# B&R Automation Studio project TD52 (part 125)

#### Ctr_HWSuCyclic.st
```iecst
(*******************************************************************************
Ctr_HWSu		controller heat water supply temperature

This code is confidential and proprietary to the INNIO Company.
It may not be used in any form, or reproduced in any manner,
without the express written permission of the INNIO Company.
Copyright, INNIO Company, 2022

Customized modifications: -
------------------------

History:
-------
V0.00.0		17.04.2012	lettenb.	Created
V3.99.0		23.11.2012	lettenb.	write back to IN_struct added (zengerer)
									tCtr_HWSu_In.Y_set := 100.0 -> 1.0, bugfix
V4.00.0		15.12.2014	lettenb.	controller interfaces completed like standard
V4.11.0		28.01.2022	Perktold	included plant controller upgrade

Instructions for use:
--------------------

Outstandings:
------------
(*******************************************************************************)

PROGRAM _CYCLIC

	(* Parameter *)
	Para.tCtr_HWSu.W_set;
	Para.tCtr_HWSu.W_set2;
	Para.tCtr_HWSu.W_min;
	Para.tCtr_HWSu.W_max;
	Para.tCtr_HWSu.dW_up;
	Para.tCtr_HWSu.dW_down;
	Para.tCtr_HWSu.deadband;
	Para.tCtr_HWSu.Y_min;
	Para.tCtr_HWSu.Y_max;
	Para.tCtr_HWSu.dY_max;
	Para.tCtr_HWSu.Y_block;
	Para.tCtr_HWSu.invert;
	Para.tCtr_HWSu.Kp;
	Para.tCtr_HWSu.Tn;
	Para.tCtr_HWSu.Tv;
	Para.tCtr_HWSu.Kp_GainScheduling;
	Para.tCtr_HWSu.Tn_GainScheduling;
	Para.tCtr_HWSu.Tv_GainScheduling;
	Para.tCtr_HWSu.t_min_pulse_down;
	Para.tCtr_HWSu.t_min_pulse_up;
	Para.tCtr_HWSu.t_period_down;
	Para.tCtr_HWSu.t_period_up;

	(* Input variables *)
	tCtr_HWSu_In				:= VIS2MM.tCtr_HWSu_In;			(* from vis *)

	(* Input from module *)
	tCtr_HWSu_In.enable			:=	Para.bCtr_HWSu
								AND	IN_HC.tPB2MM.bParaSetupOk
								AND IN_HC.bEng_Aux_Dem_CDR
								AND IN_HC.tT_HW_Su.GoodQual;
	tCtr_HWSu_In.W_ext_Active	:= tCtr_HWSu_In.W_ext_Active;	(* from vis *)
	tCtr_HWSu_In.W_ext			:= 0.0;
	tCtr_HWSu_In.Y_set_Active	:= NOT IN_HC.tT_HW_Su.GoodQual;
	tCtr_HWSu_In.Y_set			:= 1.0;
	tCtr_HWSu_In.X				:= IN_HC.tT_HW_Su.Ai;
	tCtr_HWSu_In.A				:= 0;
	tCtr_HWSu_In.W_set2_Active	:= FALSE;	(*Input to define which internal setpoint will be used TRUE = use the 2nd set point | FALSE use the normal "1st" one*)
	tCtr_HWSu_In.GainScheduling	:= 0.0;		(*Input for Gain Scheduling: 0.0 = use 100% of the Standard PID-Parameters | 1.0 = use 100% of the GainSched. PID Parameters | linear interpolation in between*)
	tCtr_HWSu_In.Y_min_cust		:= -1.0;	(*"customized" Y-Min at the current moment (The existing Y-Min parameter is the global minimum. To have an effect Y_min_cust needs to be > the parameter | -1.0 = function not used*)
	tCtr_HWSu_In.Y_max_cust		:= 1.0;		(*"customized" Y-Max at the current moment (The existing Y-Max parameter is the global maximum. To have an effect Y_max_cust needs to be < the parameter | 1.0 = function not used*)
	tCtr_HWSu_In.Retrigger		:= FALSE;	(*a rising edge on this input signals the controller to retrigger - set W on X and force the Integrator to the current Y*)

	(* Input from Visualization via OPC *)
	tCtr_HWSu_In.Y_man_Active;
	tCtr_HWSu_In.Y_man;
	tCtr_HWSu_In.X_min;
	tCtr_HWSu_In.X_max;
	tCtr_HWSu_In.Tune_quality;
	tCtr_HWSu_In.Tune_PI;
	tCtr_HWSu_In.Tune_PID;
	tCtr_HWSu_In.Tune_start;
	tCtr_HWSu_In.Tune_stop;
	tCtr_HWSu_In.Tune_takeover;

	xCtr_HWSu();

	(* Output variables function block *)
	(* Output to module(s) *)
	OUT_HC.tCtr_HWSu_Set.Ao 	:= tCtr_HWSu_Out.Y;	(* analog out *)

	(* Output to Visualization via OPC *)
	MM2VIS.tCtr_HWSu_Out		:= tCtr_HWSu_Out;
	VIS2MM.tCtr_HWSu_In			:= tCtr_HWSu_In;	(* write back to IN_struct for reset: Tune_takeover, X-display, ...!*)

	tCtr_HWSu_Out.Active;
	tCtr_HWSu_Out.Y;
	tCtr_HWSu_Out.W;
	tCtr_HWSu_Out.e;
	tCtr_HWSu_Out.Kp_tune;
	tCtr_HWSu_Out.Tn_tune;
	tCtr_HWSu_Out.Tv_tune;
	tCtr_HWSu_Out.status;

END_PROGRAM
```

#### Ctr_HWSuInit.st
```iecst
PROGRAM _INIT

	xCtr_HWSu.pParameter := ADR(Para.tCtr_HWSu);
	xCtr_HWSu.pInput 	 := ADR(tCtr_HWSu_In);
	xCtr_HWSu.pOutput	 := ADR(tCtr_HWSu_Out);

	tCtr_HWSu_In.AlwaysUseYRamp		:= TRUE;	(*If TRUE the Y signal will always limit the change rate via the according parameter | if FALSE the Y signal will jump in case the controller is disabled (blocked or set)*)
	tCtr_HWSu_In.KeepYManAtBlock	:= TRUE;	(*If TRUE the controller will keep the Y-man value constant in case the controller is disabled (blocked or set) | If FALSE the blocked or set value will override the Y-man value*)
	tCtr_HWSu_In.Y_min_cust			:= -1.0;	(*"customized" Y-Min at the current moment (The existing Y-Min parameter is the global minimum. To have an effect Y_min_cust needs to be > the parameter | -1.0 = function not used*)
	tCtr_HWSu_In.Y_max_cust			:=  1.0;	(*"customized" Y-Max at the current moment (The existing Y-Max parameter is the global maximum. To have an effect Y_max_cust needs to be < the parameter | 1.0 = function not used*)
	tCtr_HWSu_In.StepperMode		:= FALSE;	(* TRUE = use PWM-Mode (standard mode until 4.10) | FALSE = use continuous servo drive *)

END_PROGRAM
```

### Program Logical/HeatingCooling/MsgHC (IEC) - messages

#### MsgHCCyclic.st
```iecst
(*******************************************************************************
MsgHC	 			 messages

This code is confidential and proprietary to the INNIO Company.
It may not be used in any form, or reproduced in any manner,
without written permission of the INNIO Company.
Copyright, INNIO Company, 2025

Customized modifications: -
------------------------

History:
-------
V0.01.0	02.11.2011	lettenb.	new
V3.30.0 14.09.2011	lettenb.	2119 xTON_ChC_FanRdy added
V3.99.0	20.02.2013	lettenb.	3303,3521,3590 IN_HC.tT_HW_Re_LT.Ai added (V3.40)
		27.05.2013				3521 Para.bT_HW_Re_LT_Active added
		27.05.2013	Lettenb.	reset OUT_xx.txx2AB.bGnlTripx changed
		31.01.2014	lettenb.	1063 BWS_HA added(1063 NOT resetable in CASE OF sensor fail.)V350
V4.00.0	02.06.2014	lettenb.	3509 AND NOT MM2VIS.bMsg3312 added(hi-alarm in case of ms failure)
		16.06.2014	lettenb.	2104 xTP_2104, PT:= 0->1" added, acc.xt3 bugfix
V4.00.1 15.09.2014	lettenb.	1063 Para.bT_HW_Su_Active added
V4.00.2 17.11.2014				2638,2639,2640,2641,2647,2667 added, 920
								2104 enable with IN_HC.tPB2MM.bSys_Run
V4.00.3	19.03.2015				1021 STB active for 920+visa
		02.04.2015				2119 bugfix(portation failure from xt3)
V4.03.0 06.07.2015				920 ECW + EO module signals added(TCA redesign)
		25.07.2015	Plattner	2731-2736,2750,2751 failure boiler house ventilator added
		30.09.2015				2119 tAuxV_Aux_ok added
		17.03.2016	lettenb.	1021 KTMA_VISA added (920 umschaltung prio)
V4.04.0 07.04.2016	lettenb.	3492,3493,3494 added (TCA redesign2), 2640 disabled(double coded, 3590)
								2732,2734,2751 MS added + T#0s -> 2s, bugfix
		24.10.2016				2763 Functional Safety EN 13849
V4.05.0 27.02.2017	lettenb.	1032,1033 disabled for BR9 -> 2428,2429 added, SWAT920/1
		04.12.2017	Waldhart	1032,1033 enabled FOR BR9 -> 2428,2429 disabled, SWAT920/4
		22.12.2017	lettenb.	comment added: Safety-related application software source code (EN 13849-1 / 4.6.3)
		22.01.2018	lettenb.	1145,1186,1187,3407,3508,3526,3590 bParaSetupOk added TO avoid message at plc startup
V4.07.0	09.08.2018	Schmid		2nd low temperature charge cooling circuit added (W9226, W9228-W9232)
		08.10.2018	lettenb.	1063,1070,1071,1186,1187,2430,3312,3321,3508,3526,3590,9232 :bOMSS... removed, signal failure active in stop-mode
		11.10.2018	lettenb.	2720: enable Para.bT_Re_SecCirc_Active, bugfix
		17.12.2018	Schmid		OUT_HC.bMsg2684 -> AG vvm added
		06.06.2019	lettenb.	2733,2736,2752,3492,3493,3494 bParaSetupOk added to avoid alarm at plc-startup
V4.10.0	20.07.2020	Schmid		2341, 2342, 2343 additional heating water circuit monitoring
V4.11.0	17.01.2022	lettenb.	2736 delay 2s added, bugfix
V4.14.0 08.11.2024	Bacci		9098, 9099 added
		11.12.2024	Nagy		1019,1021,1050,3402 modified (2024-225)
V4.25.0	10.07.2025	Tinello		SafetyPLC: Added monitoring for heating water supply temperature unit W9588, W9589

Instructions for use:
--------------------
1) declare alarm with function block "Msg"
	declare buffert alarm bit bMsg<message number>

2) use template to create a new alarm,
   substitue 0000 by alarm number and make settings:

	xMsg0000.Enable		:=	TRUE;		enable/disable alarm
	xMsg0000.Set		:=	FALSE;		alarm set condition
	xMsg0000.PT			:=	T#0s;		alarm delay time
	xMsg0000.Prio		:=	1;			alarm priority: 1-3 = trip, 4 = warning
	xMsg0000.RiskClass	:=	3;			risk class for remote alarm reset acc.TI 1100-0111
	xMsg0000.Reset		:=	FALSE;		FALSE: for all standard alarms	prio 1,2,3 and warnings prio 4
										TRUE : for autoreset alarms

	bMsg0000			:=	xMsg0000.Q;	connect buffert alarm bit for VIS and control
	bMsg0000_Test		:=	xMsg0000.Test; alarm bypass active

3)  expand INIT

Outstandings:
------------
(*******************************************************************************)
PROGRAM _CYCLIC

	(* reset general trip *)
	OUT_HC.tHC2AB.bGnlTrip1		:=	FALSE;
	OUT_HC.tHC2AB.bGnlTrip2		:=	FALSE;
	OUT_HC.tHC2AB.bGnlTrip3		:=	FALSE;
	OUT_HC.tHC2AB.bGnlWarning	:=	FALSE;
	OUT_HC.tHC2AB.bTriptype1	:=	FALSE;
	OUT_HC.tHC2AB.bTriptype2	:=	FALSE;
	OUT_HC.tHC2AB.bTriptype3	:=	FALSE;

	(*---------------------------------------------------------------------------*)
	xTON_EngRunAnd10s(IN:= IN_HC.tEng_Run.Do, PT:= T#10s);
	xTON_EngRunAnd60s(IN:= IN_HC.tEng_Run.Do, PT:= T#60s);

	(********************************************************************************************************************
	Safety-related application software source code (EN 13849-1 / 4.6.3): BEGIN
	*********************************************************************************************************************)

	(*  1019 engine cooling water pressure low *)
	xTP_1019(IN:= IN_HC.tECWP1Dem.Do, PT:= T#10s);	(* lock monitoring *)

	xMsg1019.Enable		:=	TRUE;
	xMsg1019.Set		:=	(bPr_ECW_LoLo OR bPr_ECW_LoLoPrio2) AND NOT xTP_1019.Q;
	xMsg1019.PT			:=	T#0s;
	IF bPr_ECW_LoLoPrio2 THEN
		xMsg1019.Prio		:=	2;
	ELSE
		xMsg1019.Prio		:=	3;
	END_IF;
	xMsg1019.RiskClass	:=	10;
	xMsg1019.Reset		:=	FALSE;
	xMsg1019();
	MM2VIS.bMsg1019     := xMsg1019.Q;
	OUT_HC.bMsg1019     := xMsg1019.Q;

	(********************************************************************************************************************
	Safety-related application software source code (EN 13849-1 / 4.6.3): END
	*********************************************************************************************************************)

	(* A1021 engine cooling water temperature high *)
	xTON_1021(IN:= OUT_HC.bT_ECW_Hi, PT:= T#2h);

	xMsg1021.Enable		:=	TRUE;
	xMsg1021.Set		:= ((xTON_1021.Q OR bT_ECW_HiHi OR bT_ECW_HiHiPrio2) AND xTON_EngRunAnd60s.Q AND NOT MM2VIS.bMsg2101)
						OR  IN_HC.tT_ECW_Ext_Hi.Di; (*STB: VISA + 920*)
	xMsg1021.PT			:=	T#0s;
	KTMA_VISA := IN_HC.tT_ECW_Ext_Hi.Di OR (KTMA_VISA AND xMsg1021.Q);
	IF (Para.bVISA OR xEngType.Type9) AND KTMA_VISA OR bT_ECW_HiHiPrio2 THEN	(* umschaltung prio nur bei abstellung durch STB(sicherheitsschleife) *)
		xMsg1021.Prio	:=	2;
	ELSE
		xMsg1021.Prio	:=	3;
	END_IF;
	xMsg1021.RiskClass	:=	0;
	xMsg1021.Reset		:=	FALSE;
	xMsg1021();
	MM2VIS.bMsg1021     := xMsg1021.Q;

	(* A1032 heat water flow low (W2428)*)
	xTOF_EngDemEPS(IN:= IN_HC.bEng_Dem_EPS AND NOT IN_HC.tGCB_On.Di, PT:= T#60s);
	bNoMon4BlackStart := xTOF_EngDemEPS.Q AND IN_HC.bEng_Dem_EPS; //T14

	xMsg1032.Enable		:=	TRUE;//SWAT920/4
	xMsg1032.Set 		:=	NOT IN_HC.tFlow_HW_Lo.Di
						AND NOT bNoMon4BlackStart AND IN_HC.tEng_Run.Do;
	xMsg1032.PT			:=	T#10s;
	xMsg1032.Prio		:=	3;
	xMsg1032.RiskClass	:=	4;
	xMsg1032.Reset		:=	FALSE;
	xMsg1032();
	MM2VIS.bMsg1032     := xMsg1032.Q;

	(* A1033 heat water temperature high (W2429)*)
	xMsg1033.Enable		:=	TRUE;//SWAT920/4
	xMsg1033.Set 		:=	IN_HC.tT_HW_Hi.Di OR IN_HC.tT_HW_Hi1.Di;
	xMsg1033.PT			:=	T#0s;
	xMsg1033.Prio		:=	2;
	xMsg1033.RiskClass	:=	4;
	xMsg1033.Reset		:=	FALSE;
	xMsg1033();
	MM2VIS.bMsg1033     := xMsg1033.Q;

	(* A1034 heat water pressure low *)
	xMsg1034.Enable		:=	TRUE;
	xMsg1034.Set 		:=  IN_HC.tPr_HW_Lo.Di;
	xMsg1034.PT			:=	T#0s;
	xMsg1034.Prio		:=	2;
	xMsg1034.RiskClass	:=	4;
	xMsg1034.Reset		:=	FALSE;
	xMsg1034();
	MM2VIS.bMsg1034     := xMsg1034.Q;

	(* A1035 heat water pressure high *)
	xMsg1035.Enable		:=	TRUE;
	xMsg1035.Set 		:=  IN_HC.tPr_HW_Hi.Di OR IN_HC.tPr_HW_Hi1.Di;
	xMsg1035.PT			:=	T#0s;
	xMsg1035.Prio		:=	2;
	xMsg1035.RiskClass	:=	4;
	xMsg1035.Reset		:=	FALSE;
	xMsg1035();
	MM2VIS.bMsg1035     := xMsg1035.Q;

	(* A1050 engine cooling water pressure high *)
	(* lock monitoring jacket water pressure high at engine start. (reference: W3406)
	(in case of rising jacket water pressure with rising oil pressure.
	caused by pressure transfered from oil circuit to water circuit by the plate heat exchanger)*)
	xTP_1050(IN:= bN_EngStart, PT:= T#20s);

	xMsg1050.Enable		:=	TRUE;
	xMsg1050.Set := (bPr_ECW_HiHi OR bPr_ECW_HiHiPrio2) AND NOT xTP_1050.Q;
	xMsg1050.PT			:=	T#0s;
	IF bPr_ECW_HiHiPrio2 THEN
		xMsg1050.Prio		:=	2;
	ELSE
		xMsg1050.Prio		:=	3;
	END_IF;
	xMsg1050.RiskClass	:=	2;
	xMsg1050.Reset		:=	FALSE;
	xMsg1050();
	MM2VIS.bMsg1050     := xMsg1050.Q;
	OUT_HC.bMsg1050		:= xMsg1050.Q;

	(* A1063 heat water supply temperature high (W2430)*)
	xMsg1063.Enable		:=	Para.bT_HW_Su_Active;
	xMsg1063.Set 		:=  bT_HW_Su_HiHi AND NOT MM2VIS.bMsg1071 AND NOT MM2VIS.bMsg1187;
	xMsg1063.PT			:=	T#2s;
	xMsg1063.Prio		:=	3;
	xMsg1063.RiskClass	:=	0;
	xMsg1063.Reset		:=	FALSE;
	xMsg1063();
	MM2VIS.bMsg1063     := xMsg1063.Q;

	(* A1070 heat water return temperature signal failure trip (W1186)*)
	xMsg1070.Enable		:=	Para.bT_HW_Re_Active AND Para.bT_HW_Re_SF_Trip;
	xMsg1070.Set 		:=	NOT IN_HC.tT_HW_Re.GoodQual;
	xMsg1070.PT			:=	T#0s;
	xMsg1070.Prio		:=	3;
	xMsg1070.RiskClass	:=	4;
	xMsg1070.Reset		:=	FALSE;
	xMsg1070();
	MM2VIS.bMsg1070     := xMsg1070.Q;

	(* A1071 heat water supply temperature signal failure trip (W1187)*)
	xMsg1071.Enable		:=	Para.bT_HW_Su_Active AND Para.bT_HW_Su_SF_Trip;
	xMsg1071.Set 		:=  NOT IN_HC.tT_HW_Su.GoodQual;
	xMsg1071.PT			:=	T#0s;
	xMsg1071.Prio		:=	3;
	xMsg1071.RiskClass	:=	4;
	xMsg1071.Reset		:=	FALSE;
	xMsg1071();
	MM2VIS.bMsg1071     := xMsg1071.Q;

	(* A1130 charge cooler water pressure low (W2117)*)
	xMsg1130.Enable		:=	FALSE;
	xMsg1130.Set		:=	NOT IN_HC.tPr_ChC_Lo.Di;
	xMsg1130.PT			:=	T#0s;
	xMsg1130.Prio		:=	3;
	xMsg1130.RiskClass	:=	4;
	xMsg1130.Reset		:=	FALSE;
	xMsg1130();
	MM2VIS.bMsg1130     := xMsg1130.Q;

	(* W1145 engine cooling water temperature low *)
	xMsg1145.Enable		:=	IN_HC.tPB2MM.bParaSetupOk;
	xMsg1145.Set 		:=  OUT_HC.bT_ECW_Lo;
	xMsg1145.PT			:=	T#0s;
	xMsg1145.Prio		:=	4;
	xMsg1145.RiskClass	:=	4;
	xMsg1145.Reset		:=	FALSE;
	xMsg1145();
	MM2VIS.bMsg1145     := xMsg1145.Q;

	(* W1167  heat water return temperature high *)
	xTON_1167(IN:= NOT MM2VIS.bMsg1186 AND NOT MM2VIS.bMsg1070 AND bT_HW_Re_Hi, PT:= T#10s);

	xMsg1167.Enable		:=	Para.bT_HW_Re_Active;
	xMsg1167.Set 		:=  xTON_EngRunAnd10s.Q AND xTON_1167.Q;
	xMsg1167.PT			:=	T#0s;
	xMsg1167.Prio		:=	4;
	xMsg1167.RiskClass	:=	4;
	xMsg1167.Reset		:=	FALSE;
	xMsg1167();
	MM2VIS.bMsg1167     := xMsg1167.Q;

	(* W1186 heat water return temperature signal failure (A1070)*)
	xMsg1186.Enable		:=	Para.bT_HW_Re_Active AND NOT Para.bT_HW_Re_SF_Trip AND IN_HC.tPB2MM.bParaSetupOk;
	xMsg1186.Set 		:=  NOT IN_HC.tT_HW_Re.GoodQual;
	xMsg1186.PT			:=	T#0s;
	xMsg1186.Prio		:=	4;
	xMsg1186.RiskClass	:=	4;
	xMsg1186.Reset		:=	FALSE;
	xMsg1186();
	MM2VIS.bMsg1186     := xMsg1186.Q;

	(* W1187 heat water supply temperature signal failure (A1071)*)
	xMsg1187.Enable		:=	Para.bT_HW_Su_Active AND NOT Para.bT_HW_Su_SF_Trip AND IN_HC.tPB2MM.bParaSetupOk;
	xMsg1187.Set 		:=  NOT IN_HC.tT_HW_Su.GoodQual;
	xMsg1187.PT			:=	T#0s;
	xMsg1187.Prio		:=	4;
	xMsg1187.RiskClass	:=	4;
	xMsg1187.Reset		:=	FALSE;
	xMsg1187();
	MM2VIS.bMsg1187     := xMsg1187.Q;

	(* W2101 engine cooling water temperature signal failure *)
	xMsg2101.Enable		:=	TRUE;
	xMsg2101.Set		:= (NOT IN_HC.tT_ECW.GoodQual AND IN_HC.tPB2MM.bParaSetupOk)
						OR (xMsg2101.Set AND IN_HC.bMsg3003 AND bOMSS_MAT);
	xMsg2101.PT			:=	T#0s;
	xMsg2101.Prio		:=	4;
	xMsg2101.RiskClass	:=	4;
	xMsg2101.Reset		:=	FALSE;
	xMsg2101();
	MM2VIS.bMsg2101     := xMsg2101.Q;
	OUT_HC.bMsg2101     := xMsg2101.Q;

	(********************************************************************************************************************
	Safety-related application software source code (EN 13849-1 / 4.6.3): BEGIN
	*********************************************************************************************************************)
	(* W2104 engine cooling water pressure signal failure *)
	xTP_2104(IN:= IN_HC.tECWP1Dem.Do, PT:= T#10s);	(* lock monitoring *)

	xMsg2104.Enable		:=	IN_HC.tPB2MM.bSys_Run;
	xMsg2104.Set		:= (NOT IN_HC.tPr_ECW.GoodQual AND NOT xTP_2104.Q)
						OR (xMsg2104.Set AND IN_HC.bMsg3003 AND bOMSS_MAT);
	xMsg2104.PT			:=	T#1s;
	xMsg2104.Prio		:=	4;
	xMsg2104.RiskClass	:=	4;
	xMsg2104.Reset		:=	FALSE;
	xMsg2104();
	MM2VIS.bMsg2104     := xMsg2104.Q;
	OUT_HC.bMsg2104     := xMsg2104.Q;
	(********************************************************************************************************************
	Safety-related application software source code (EN 13849-1 / 4.6.3): END
	*********************************************************************************************************************)

	(* W2116 emergency cooler failure *)
	xMsg2116.Enable		:=	TRUE;
	xMsg2116.Set		:=	NOT IN_HC.tEC_Failure.Di AND NOT bNoMon4BlackStart;
	xMsg2116.PT			:=	T#0s;
	xMsg2116.Prio		:=	4;
	xMsg2116.RiskClass	:=	4;
	xMsg2116.Reset		:=	FALSE;
	xMsg2116();
	MM2VIS.bMsg2116     := xMsg2116.Q;

	(* W2117 charge cooler water pressure low (A1130)*)
	xMsg2117.Enable		:=	TRUE;
	xMsg2117.Set		:=	NOT IN_HC.tPr_ChC_Lo.Di;
	xMsg2117.PT			:=	T#10s;
	xMsg2117.Prio		:=	4;
	xMsg2117.RiskClass	:=	4;
	xMsg2117.Reset		:=	FALSE;
	xMsg2117();
	MM2VIS.bMsg2117     := xMsg2117.Q;
	OUT_HC.bMsg2117     := xMsg2117.Q;

	(* W2119 charge cooler failure *)
	xTON_ChC_FanRdy(IN:= (IN_HC.tAuxV_Supply_Ok.Di AND IN_HC.tAuxV_Aux_ok.Di) AND NOT IN_HC.tChC_FanRdy.Di, PT:= T#10s);		(*PJ*)

	xMsg2119.Enable		:=	TRUE;
	xMsg2119.Set		:=	NOT bNoMon4BlackStart AND(xTON_ChC_FanRdy.Q OR NOT IN_HC.tChC_Failure.Di);
	xMsg2119.PT			:=	T#0s;
	xMsg2119.Prio		:=	4;
	xMsg2119.RiskClass	:=	4;
	xMsg2119.Reset		:=	FALSE;
	xMsg2119();
	MM2VIS.bMsg2119     := xMsg2119.Q;

	(* A2341 Heating water temperature maximum - exhaust gas cooler *)
	xMsg2341.Enable		:=	IN_HC.tT_HW_EGHE_Hi.GoodQual;
	xMsg2341.Set 		:=	IN_HC.tT_HW_EGHE_Hi.Di;
	xMsg2341.PT			:=	T#0s;
	xMsg2341.Prio		:=	2;
	xMsg2341.RiskClass	:=	4;
	xMsg2341.Reset		:=	FALSE;
	xMsg2341();
	MM2VIS.bMsg2341     := xMsg2341.Q;

	(* A2342 Heating water temperature maximum - exhaust gas condenser *)
	xMsg2342.Enable		:=	IN_HC.tT_HW_EGCD_Hi.GoodQual;
	xMsg2342.Set 		:=	IN_HC.tT_HW_EGCD_Hi.Di;
	xMsg2342.PT			:=	T#0s;
	xMsg2342.Prio		:=	2;
	xMsg2342.RiskClass	:=	4;
	xMsg2342.Reset		:=	FALSE;
	xMsg2342();
	MM2VIS.bMsg2342     := xMsg2342.Q;

	(* A2343 External heating water circuit monitoring tripped *)
	xMsg2343.Enable		:=	IN_HC.tCust_HW_Ext_Trip.GoodQual;
	xMsg2343.Set 		:=	IN_HC.tCust_HW_Ext_Trip.Di;
	xMsg2343.PT			:=	T#0s;
	xMsg2343.Prio		:=	2;
	xMsg2343.RiskClass	:=	4;
	xMsg2343.Reset		:=	FALSE;
	xMsg2343();
	MM2VIS.bMsg2343     := xMsg2343.Q;

	(* W2428 heat water flow low (A1032)*)
	xMsg2428.Enable		:=	FALSE;//SWAT920/4
	xMsg2428.Set 		:=	NOT IN_HC.tFlow_HW_Lo.Di
						AND NOT bNoMon4BlackStart AND IN_HC.tEng_Run.Do;
	xMsg2428.PT			:=	T#10s;
	xMsg2428.Prio		:=	4;
	xMsg2428.RiskClass	:=	4;
	xMsg2428.Reset		:=	FALSE;
	xMsg2428();
	MM2VIS.bMsg2428     := xMsg2428.Q;

	(* W2429 heat water temperature high (A1033)*)
	xMsg2429.Enable		:=	FALSE;//SWAT920/4
	xMsg2429.Set 		:=	IN_HC.tT_HW_Hi.Di OR IN_HC.tT_HW_Hi1.Di;
	xMsg2429.PT			:=	T#0s;
	xMsg2429.Prio		:=	4;
	xMsg2429.RiskClass	:=	4;
	xMsg2429.Reset		:=	FALSE;
	xMsg2429();
	MM2VIS.bMsg2429     := xMsg2429.Q;

	(* W2430 heat water supply temperature high (A1063)*)//SWAT920/1
	xMsg2430.Enable		:=	Para.bT_HW_Su_Active;
	xMsg2430.Set 		:=  bT_HW_Su_Hi AND NOT MM2VIS.bMsg1071 AND NOT MM2VIS.bMsg1187;
	xMsg2430.PT			:=	T#2s;
	xMsg2430.Prio		:=	4;
	xMsg2430.RiskClass	:=	0;
	xMsg2430.Reset		:=	FALSE;
	xMsg2430();
	MM2VIS.bMsg2430     := xMsg2430.Q;

	(* W2638 heat water supply pressure LT circuit signal failure *)
	xMsg2638.Enable		:=	Para.bPr_HW_Su_LT_Active;
	xMsg2638.Set		:=	IN_HC.tPB2MM.bParaSetupOk AND NOT IN_HC.tPr_HW_Su_LT.GoodQual;
	xMsg2638.PT			:=	T#0s;
	xMsg2638.Prio		:=	4;
	xMsg2638.RiskClass	:=	4;
	xMsg2638.Reset		:=	FALSE;
	xMsg2638();
	MM2VIS.bMsg2638     := xMsg2638.Q;

	(* W2639 heat water supply pressure HT circuit signal failure *)
	xMsg2639.Enable		:=	Para.bPr_HW_Su_HT_Active;
	xMsg2639.Set		:=	IN_HC.tPB2MM.bParaSetupOk AND NOT IN_HC.tPr_HW_Su_HT.GoodQual;
	xMsg2639.PT			:=	T#0s;
	xMsg2639.Prio		:=	4;
	xMsg2639.RiskClass	:=	4;
	xMsg2639.Reset		:=	FALSE;
	xMsg2639();
	MM2VIS.bMsg2639     := xMsg2639.Q;

	(* W2640 heat water return temperature LT circuit signal failure *)(* -> 3590 *)
	xMsg2640.Enable		:=	Para.bT_HW_Re_LT_Active AND FALSE;
	xMsg2640.Set		:=	IN_HC.tPB2MM.bParaSetupOk AND NOT IN_HC.tT_HW_Re_LT.GoodQual;
	xMsg2640.PT			:=	T#0s;
	xMsg2640.Prio		:=	4;
	xMsg2640.RiskClass	:=	4;
	xMsg2640.Reset		:=	FALSE;
	xMsg2640();
	MM2VIS.bMsg2640     := xMsg2640.Q;

	(* W2641 heat water supply temperature LT circuit signal failure *)
	xMsg2641.Enable		:=	Para.bT_HW_Su_LT_Active;
	xMsg2641.Set		:=	IN_HC.tPB2MM.bParaSetupOk AND NOT IN_HC.tT_HW_Su_LT.GoodQual;
	xMsg2641.PT			:=	T#0s;
	xMsg2641.Prio		:=	4;
	xMsg2641.RiskClass	:=	4;
	xMsg2641.Reset		:=	FALSE;
	xMsg2641();
	MM2VIS.bMsg2641     := xMsg2641.Q;

	(* W2647 engine cooling water pressure after engine signal failure *)
	xMsg2647.Enable	   := Para.bPr_ECWaEng_Active;
	xMsg2647.Set       := IN_HC.tPB2MM.bParaSetupOk AND NOT IN_HC.tPr_ECWaEng.GoodQual;
	xMsg2647.PT		   := T#0s;
	xMsg2647.Prio	   := 4;
	xMsg2647.RiskClass := 4;
	xMsg2647.Reset	   := FALSE;
	xMsg2647();
	MM2VIS.bMsg2647	   := xMsg2647.Q;

	(* W2667 engine cooling water temperature before engine signal failure *)
	xMsg2667.Enable	   := Para.bT_ECWbEng_Active;
	xMsg2667.Set       := IN_HC.tPB2MM.bParaSetupOk AND NOT IN_HC.tT_ECWbEng.GoodQual;
	xMsg2667.PT		   := T#0s;
	xMsg2667.Prio	   := 4;
	xMsg2667.RiskClass := 4;
	xMsg2667.Reset	   := FALSE;
	xMsg2667();
	MM2VIS.bMsg2667	   := xMsg2667.Q;

	(* W2675 Pressure heat water return low temperature circuit return signal failure *)
	xMsg2675.Enable	   := Para.bPr_HW_Re_LT_Active;
	xMsg2675.Set       := IN_HC.tPB2MM.bParaSetupOk AND NOT IN_HC.tPr_HW_Re_LT.GoodQual;
	xMsg2675.PT		   := T#0s;
	xMsg2675.Prio	   := 4;
	xMsg2675.RiskClass := 4;
	xMsg2675.Reset	   := FALSE;
	xMsg2675();
	MM2VIS.bMsg2675	   := xMsg2675.Q;

	(* W2676 Pressure heat water return high temperature circuit signal failure *)
	xMsg2676.Enable	   := Para.bPr_HW_Re_HT_Active;
	xMsg2676.Set       := IN_HC.tPB2MM.bParaSetupOk AND NOT IN_HC.tPr_HW_Re_HT.GoodQual;
	xMsg2676.PT		   := T#0s;
	xMsg2676.Prio	   := 4;
	xMsg2676.RiskClass := 4;
	xMsg2676.Reset	   := FALSE;
	xMsg2676();
	MM2VIS.bMsg2676	   := xMsg2676.Q;

	(* W2677 Pressure heat water return hydraulic engine cooling water preheating signal failure *)
	xMsg2677.Enable	   := Para.bPr_HW_Re_PreH_ECW_Active;
	xMsg2677.Set       := IN_HC.tPB2MM.bParaSetupOk AND NOT IN_HC.tPr_HW_Re_PreH_ECW.GoodQual;
	xMsg2677.PT		   := T#0s;
	xMsg2677.Prio	   := 4;
	xMsg2677.RiskClass := 4;
	xMsg2677.Reset	   := FALSE;
	xMsg2677();
	MM2VIS.bMsg2677	   := xMsg2677.Q;

	(* W2678 Pressure heat water return hydraulic oil preheating signal failure *)
	xMsg2678.Enable	   := Para.bPr_HW_Re_PreH_EO_Active;
	xMsg2678.Set       := IN_HC.tPB2MM.bParaSetupOk AND NOT IN_HC.tPr_HW_Re_PreH_EO.GoodQual;
	xMsg2678.PT		   := T#0s;
	xMsg2678.Prio	   := 4;
	xMsg2678.RiskClass := 4;
	xMsg2678.Reset	   := FALSE;
	xMsg2678();
	MM2VIS.bMsg2678	   := xMsg2678.Q;

	(* W2679 Pressure oil module oil outlet signal failure *)
	xMsg2679.Enable	   := Para.bPr_EO_Mod_Out_Active;
	xMsg2679.Set       := IN_HC.tPB2MM.bParaSetupOk AND NOT IN_HC.tPr_EO_Mod_Out.GoodQual;
	xMsg2679.PT		   := T#0s;
	xMsg2679.Prio	   := 4;
	xMsg2679.RiskClass := 4;
	xMsg2679.Reset	   := FALSE;
	xMsg2679();
	MM2VIS.bMsg2679	   := xMsg2679.Q;

	(* W2680 Temperature engine cooling water module inlet  signal failure *)
	xMsg2680.Enable	   := Para.bT_ECW_Mod_In_Active;
	xMsg2680.Set       := IN_HC.tPB2MM.bParaSetupOk AND NOT IN_HC.tT_ECW_Mod_In.GoodQual;
	xMsg2680.PT		   := T#0s;
	xMsg2680.Prio	   := 4;
	xMsg2680.RiskClass := 4;
	xMsg2680.Reset	   := FALSE;
	xMsg2680();
	MM2VIS.bMsg2680	   := xMsg2680.Q;

	(* W2681 Temperature engine cooling water module outlet  signal failure *)
	xMsg2681.Enable	   := Para.bT_ECW_Mod_Out_Active;
	xMsg2681.Set       := IN_HC.tPB2MM.bParaSetupOk AND NOT IN_HC.tT_ECW_Mod_Out.GoodQual;
	xMsg2681.PT		   := T#0s;
	xMsg2681.Prio	   := 4;
	xMsg2681.RiskClass := 4;
	xMsg2681.Reset	   := FALSE;
	xMsg2681();
	MM2VIS.bMsg2681	   := xMsg2681.Q;

	(* W2682 Temperature oil module oil inlet signal failure *)
	xMsg2682.Enable	   := Para.bT_EO_Mod_In_Active;
	xMsg2682.Set       := IN_HC.tPB2MM.bParaSetupOk AND NOT IN_HC.tT_EO_Mod_In.GoodQual;
	xMsg2682.PT		   := T#0s;
	xMsg2682.Prio	   := 4;
	xMsg2682.RiskClass := 4;
	xMsg2682.Reset	   := FALSE;
	xMsg2682();
	MM2VIS.bMsg2682	   := xMsg2682.Q;

	(* W2683 Temperature oil module oil outlet  signal failure *)
	xMsg2683.Enable	   := Para.bT_EO_Mod_Out_Active;
	xMsg2683.Set       := IN_HC.tPB2MM.bParaSetupOk AND NOT IN_HC.tT_EO_Mod_Out.GoodQual;
	xMsg2683.PT		   := T#0s;
	xMsg2683.Prio	   := 4;
	xMsg2683.RiskClass := 4;
	xMsg2683.Reset	   := FALSE;
	xMsg2683();
	MM2VIS.bMsg2683	   := xMsg2683.Q;

	(* W2684 Temperature heat water supply hydraulic engine cooling water preheating signal failure *)
	xMsg2684.Enable	   := Para.bT_HW_Su_PreH_ECW_Active;
	xMsg2684.Set       := IN_HC.tPB2MM.bParaSetupOk AND NOT IN_HC.tT_HW_Su_PreH_ECW.GoodQual;
	xMsg2684.PT		   := T#0s;
	xMsg2684.Prio	   := 4;
	xMsg2684.RiskClass := 4;
	xMsg2684.Reset	   := FALSE;
	xMsg2684();
	MM2VIS.bMsg2684	   := xMsg2684.Q;
	OUT_HC.bMsg2684    := xMsg2684.Q;

	(* W2685 Temperature heat water return hydraulic engine cooling water preheating signal failure *)
	xMsg2685.Enable	   := Para.bT_HW_Re_PreH_ECW_Active;
	xMsg2685.Set       := IN_HC.tPB2MM.bParaSetupOk AND NOT IN_HC.tT_HW_Re_PreH_ECW.GoodQual;
	xMsg2685.PT		   := T#0s;
	xMsg2685.Prio	   := 4;
	xMsg2685.RiskClass := 4;
	xMsg2685.Reset	   := FALSE;
	xMsg2685();
	MM2VIS.bMsg2685	   := xMsg2685.Q;

	(* W2686 Temperature heat water supply hydraulic oil preheating signal failure *)
	xMsg2686.Enable	   := Para.bT_HW_Su_PreH_EO_Active;
	xMsg2686.Set       := IN_HC.tPB2MM.bParaSetupOk AND NOT IN_HC.tT_HW_Su_PreH_EO.GoodQual;
	xMsg2686.PT		   := T#0s;
	xMsg2686.Prio	   := 4;
	xMsg2686.RiskClass := 4;
	xMsg2686.Reset	   := FALSE;
	xMsg2686();
	MM2VIS.bMsg2686	   := xMsg2686.Q;

	(* W2687 Temperature heat water return hydraulic oil preheating signal failure *)
	xMsg2687.Enable	   := Para.bT_HW_Re_PreH_EO_Active;
	xMsg2687.Set       := IN_HC.tPB2MM.bParaSetupOk AND NOT IN_HC.tT_HW_Re_PreH_EO.GoodQual;
	xMsg2687.PT		   := T#0s;
	xMsg2687.Prio	   := 4;
	xMsg2687.RiskClass := 4;
	xMsg2687.Reset	   := FALSE;
	xMsg2687();
	MM2VIS.bMsg2687	   := xMsg2687.Q;

	(* W2710 measuring signal failure position control valve heat water return temperature *)
	xMsg2710.Enable		:=	Para.bPos_HW_ReValve;
	xMsg2710.Set 		:= 	IN_HC.tPB2MM.bParaSetupOk AND NOT IN_HC.tPos_HW_ReValve.GoodQual;
	xMsg2710.PT			:=	T#0s;
	xMsg2710.Prio		:=	4;
	xMsg2710.RiskClass	:=	4;
	xMsg2710.Reset		:=	FALSE;
	xMsg2710();
	MM2VIS.bMsg2710     := xMsg2710.Q;

	(* W2711 measuring signal failure position control valve heat water return temperature after cooler *)
	xMsg2711.Enable		:=	Para.bPos_HW_EC_ReValve;
	xMsg2711.Set 		:= 	IN_HC.tPB2MM.bParaSetupOk AND NOT IN_HC.tPos_HW_EC_ReValve.GoodQual;
	xMsg2711.PT			:=	T#0s;
	xMsg2711.Prio		:=	4;
	xMsg2711.RiskClass	:=	4;
	xMsg2711.Reset		:=	FALSE;
	xMsg2711();
	MM2VIS.bMsg2711     := xMsg2711.Q;

	(* W2712 measuring signal failure position control valve charge cooler circuit temperature *)
	xMsg2712.Enable		:=	Para.bPos_ChCValve;
	xMsg2712.Set 		:= 	IN_HC.tPB2MM.bParaSetupOk AND NOT IN_HC.tPos_ChC_Valve.GoodQual;
	xMsg2712.PT			:=	T#0s;
	xMsg2712.Prio		:=	4;
	xMsg2712.RiskClass	:=	4;
	xMsg2712.Reset		:=	FALSE;
	xMsg2712();
	MM2VIS.bMsg2712     := xMsg2712.Q;

	(* W2713 measuring signal failure supply water temperature primary circuit *)
	xMsg2713.Enable		:=	Para.bT_Su_PriCirc_Active;
	xMsg2713.Set 		:= 	IN_HC.tPB2MM.bParaSetupOk AND NOT IN_HC.tT_Su_PriCirc.GoodQual;
	xMsg2713.PT			:=	T#0s;
	xMsg2713.Prio		:=	4;
	xMsg2713.RiskClass	:=	4;
	xMsg2713.Reset		:=	FALSE;
	xMsg2713();
	MM2VIS.bMsg2713     := xMsg2713.Q;

	(* W2714 measuring signal failure return water temperature primary circuit *)
	xMsg2714.Enable		:=	Para.bT_Re_PriCirc_Active;
	xMsg2714.Set 		:= 	IN_HC.tPB2MM.bParaSetupOk AND NOT IN_HC.tT_Re_PriCirc.GoodQual;
	xMsg2714.PT			:=	T#0s;
	xMsg2714.Prio		:=	4;
	xMsg2714.RiskClass	:=	4;
	xMsg2714.Reset		:=	FALSE;
	xMsg2714();
	MM2VIS.bMsg2714     := xMsg2714.Q;

	(* W2715 measuring signal failure supply water temperature secondary circuit *)
	xMsg2715.Enable		:=	Para.bT_Su_SecCirc_Active;
	xMsg2715.Set 		:= 	IN_HC.tPB2MM.bParaSetupOk AND NOT IN_HC.tT_Su_SecCirc.GoodQual;
	xMsg2715.PT			:=	T#0s;
	xMsg2715.Prio		:=	4;
	xMsg2715.RiskClass	:=	4;
	xMsg2715.Reset		:=	FALSE;
	xMsg2715();
	MM2VIS.bMsg2715     := xMsg2715.Q;

	(* W2716 measuring signal failure return water temperature secondary circuit *)
	xMsg2716.Enable		:=	Para.bT_Re_SecCirc_Active;
	xMsg2716.Set 		:= 	IN_HC.tPB2MM.bParaSetupOk AND NOT IN_HC.tT_Re_SecCirc.GoodQual;
	xMsg2716.PT			:=	T#0s;
	xMsg2716.Prio		:=	4;
	xMsg2716.RiskClass	:=	4;
	xMsg2716.Reset		:=	FALSE;
	xMsg2716();
	MM2VIS.bMsg2716     := xMsg2716.Q;

	(* W2717 supply water temperature high primary circuit *)
	xGRMAX_T_Su_PriCirc(In:= IN_HC.tT_Su_PriCirc.Ai, Gw:= Para.rT_Su_PriCirc_LimHi, Hy:= Para.rT_Su_PriCirc_HyLimHi);
	bT_Su_PriCirc_Hi := xGRMAX_T_Su_PriCirc.Q;

	xMsg2717.Enable		:=	Para.bT_Su_PriCirc_Active;
	xMsg2717.Set 		:= 	bT_Su_PriCirc_Hi AND NOT MM2VIS.bMsg2713;
	xMsg2717.PT			:=	T#0s;
	xMsg2717.Prio		:=	4;
	xMsg2717.RiskClass	:=	4;
	xMsg2717.Reset		:=	FALSE;
	xMsg2717();
	MM2VIS.bMsg2717     := xMsg2717.Q;

	(* W2718 return water temperature high primary circuit *)
	xGRMAX_T_Re_PriCirc(In:= IN_HC.tT_Re_PriCirc.Ai, Gw:= Para.rT_Re_PriCirc_LimHi, Hy:= Para.rT_Re_PriCirc_HyLimHi);
	bT_Re_PriCirc_Hi := xGRMAX_T_Re_PriCirc.Q;

	xMsg2718.Enable		:=	Para.bT_Re_PriCirc_Active;
	xMsg2718.Set 		:= 	bT_Re_PriCirc_Hi AND NOT MM2VIS.bMsg2714;
	xMsg2718.PT			:=	T#0s;
	xMsg2718.Prio		:=	4;
	xMsg2718.RiskClass	:=	4;
	xMsg2718.Reset		:=	FALSE;
	xMsg2718();
	MM2VIS.bMsg2718     := xMsg2718.Q;

	(* W2719 supply water temperature high secondary circuit *)
	xGRMAX_T_Su_SecCirc(In:= IN_HC.tT_Su_SecCirc.Ai, Gw:= Para.rT_Su_SecCirc_LimHi, Hy:= Para.rT_Su_SecCirc_HyLimHi);
	bT_Su_SecCirc_Hi := xGRMAX_T_Su_SecCirc.Q;

	xMsg2719.Enable		:=	Para.bT_Su_SecCirc_Active;
	xMsg2719.Set 		:= 	bT_Su_SecCirc_Hi AND NOT MM2VIS.bMsg2715;
	xMsg2719.PT			:=	T#0s;
	xMsg2719.Prio		:=	4;
	xMsg2719.RiskClass	:=	4;
	xMsg2719.Reset		:=	FALSE;
	xMsg2719();
	MM2VIS.bMsg2719     := xMsg2719.Q;

	(* W2720 return water temperature high secondary circuit *)
	xGRMAX_T_Re_SecCirc(In:= IN_HC.tT_Re_SecCirc.Ai, Gw:= Para.rT_Re_SecCirc_LimHi, Hy:= Para.rT_Re_SecCirc_HyLimHi);
	bT_Re_SecCirc_Hi := xGRMAX_T_Re_SecCirc.Q;

	xMsg2720.Enable		:=	Para.bT_Re_SecCirc_Active;
	xMsg2720.Set 		:= 	bT_Re_SecCirc_Hi AND NOT MM2VIS.bMsg2716;
	xMsg2720.PT			:=	T#0s;
	xMsg2720.Prio		:=	4;
	xMsg2720.RiskClass	:=	4;
	xMsg2720.Reset		:=	FALSE;
	xMsg2720();
	MM2VIS.bMsg2720     := xMsg2720.Q;

	(* W2721 measuring signal failure heating power engine heat water circuit *)
	xMsg2721.Enable		:=	Para.bP_Heat_Active;
	xMsg2721.Set 		:= 	NOT IN_HC.tP_Heat.GoodQual;
	xMsg2721.PT			:=	T#0s;
	xMsg2721.Prio		:=	4;
	xMsg2721.RiskClass	:=	4;
	xMsg2721.Reset		:=	FALSE;
	xMsg2721();
	MM2VIS.bMsg2721     := xMsg2721.Q;

	(* W2731 measuring signal failure condensor circuit supply temperature *)
	xMsg2731.Enable		:=	Para.bT_CD_Su_Active;
	xMsg2731.Set 		:= 	NOT IN_HC.tT_CD_Su.GoodQual;
	xMsg2731.PT			:=	T#0s;
	xMsg2731.Prio		:=	4;
	xMsg2731.RiskClass	:=	4;
	xMsg2731.Reset		:=	FALSE;
	xMsg2731();
	MM2VIS.bMsg2731     := xMsg2731.Q;

	(* W2732 supply temperature condensor circuit maximum *)
	xMsg2732.Enable		:=	Para.bT_CD_Su_Active;
	xMsg2732.Set 		:= 	bT_CD_Su_Hi AND NOT MM2VIS.bMsg2731;
	xMsg2732.PT			:=	T#2s;
	xMsg2732.Prio		:=	4;
	xMsg2732.RiskClass	:=	4;
	xMsg2732.Reset		:=	FALSE;
	xMsg2732();
	MM2VIS.bMsg2732     := xMsg2732.Q;

	(* W2733 measuring signal failure return temperature condensor circuit *)
	xMsg2733.Enable		:=	Para.bT_CD_Re_Active;
	xMsg2733.Set 		:= 	IN_HC.tPB2MM.bParaSetupOk AND NOT IN_HC.tT_CD_Re.GoodQual;
	xMsg2733.PT			:=	T#0s;
	xMsg2733.Prio		:=	4;
	xMsg2733.RiskClass	:=	4;
	xMsg2733.Reset		:=	FALSE;
	xMsg2733();
	MM2VIS.bMsg2733     := xMsg2733.Q;

	(* W2734 return temperature condensor circuit maximum *)
	xMsg2734.Enable		:=	Para.bT_CD_Re_Active;
	xMsg2734.Set 		:= 	bT_CD_Re_Hi AND NOT MM2VIS.bMsg2733;
	xMsg2734.PT			:=	T#2s;
	xMsg2734.Prio		:=	4;
	xMsg2734.RiskClass	:=	4;
	xMsg2734.Reset		:=	FALSE;
	xMsg2734();
	MM2VIS.bMsg2734     := xMsg2734.Q;

	(* W2735 failure condensor pump *)
	xTOF_CDP_Fail(IN:= IN_HC.tCDP_Op.Di OR bNoMon4BlackStart, PT:= T#10s);
	HBT_1 := xTOF_CDP_Fail.Q OR (IN_HC.tCDP_Dem.Do AND HBT_1);
	xTON_CDP_Fail(IN:= IN_HC.tCDP_Dem.Do, PT:= T#175s);

	xMsg2735.Enable		:=	TRUE;
	xMsg2735.Set 		:= 	(xTON_CDP_Fail.Q OR HBT_1) AND NOT xTOF_CDP_Fail.Q;
	xMsg2735.PT			:=	T#0s;
	xMsg2735.Prio		:=	4;
	xMsg2735.RiskClass	:=	4;
	xMsg2735.Reset		:=	FALSE;
	xMsg2735();
	MM2VIS.bMsg2735     := xMsg2735.Q;

	(* W2736 failure boiler house ventilation*)
	xMsg2736.Enable		:=	TRUE;
	xMsg2736.Set 		:= 	IN_HC.tPB2MM.bParaSetupOk AND bFail_BHV;
	xMsg2736.PT			:=	T#2s;
	xMsg2736.Prio		:=	4;
	xMsg2736.RiskClass	:=	4;
	xMsg2736.Reset		:=	FALSE;
	xMsg2736();
	MM2VIS.bMsg2736     := xMsg2736.Q;

	(* W2750 failure heating circuit flap *)
	xMsg2750.Enable		:=	TRUE;
	xMsg2750.Set 		:= 	NOT IN_HC.tHWF_Fail.Di;
	xMsg2750.PT			:=	T#0s;
	xMsg2750.Prio		:=	4;
	xMsg2750.RiskClass	:=	4;
	xMsg2750.Reset		:=	FALSE;
	xMsg2750();
	MM2VIS.bMsg2750     := xMsg2750.Q;

	(* W2751 heat circuit return temperature high *)
	xMsg2751.Enable		:=	TRUE;
	xMsg2751.Set 		:= 	bT_HW_HC_Re_Hi AND NOT MM2VIS.bMsg2752;
	xMsg2751.PT			:=	T#2s;
	xMsg2751.Prio		:=	4;
	xMsg2751.RiskClass	:=	4;
	xMsg2751.Reset		:=	FALSE;
	xMsg2751();
	MM2VIS.bMsg2751     := xMsg2751.Q;

	(* W2752 signal failur heat circuit return temperature *)
	xMsg2752.Enable		:=	Para.bT_HW_HC_Re_Active;
	xMsg2752.Set 		:= 	IN_HC.tPB2MM.bParaSetupOk AND NOT IN_HC.tT_HW_HC_Re.GoodQual;
	xMsg2752.PT			:=	T#0s;
	xMsg2752.Prio		:=	4;
	xMsg2752.RiskClass	:=	4;
	xMsg2752.Reset		:=	FALSE;
	xMsg2752();
	MM2VIS.bMsg2752     := xMsg2752.Q;

	(********************************************************************************************************************
	Safety-related application software source code (EN 13849-1 / 4.6.3): BEGIN
	*********************************************************************************************************************)
	(* W2763 plausibility check measuring signal engine cooling water pressure (Functional Safety) *)
	xMsg2763.Enable		:=	IN_HC.tPB2MM.bSys_Run;
	xMsg2763.Set 		:= 	bPr_ECW_PcheckFail;
	xMsg2763.PT			:=	T#0s;
	xMsg2763.Prio		:=	4;
	xMsg2763.RiskClass	:=	4;
	xMsg2763.Reset		:=	FALSE;
	xMsg2763();
	MM2VIS.bMsg2763     := xMsg2763.Q;
	(********************************************************************************************************************
	Safety-related application software source code (EN 13849-1 / 4.6.3): END
	*********************************************************************************************************************)

	(* W3220 engine cooling water temperature high *)
	xMsg3220.Enable		:=	TRUE;
	xMsg3220.Set		:=	OUT_HC.bT_ECW_Hi AND xTON_EngRunAnd60s.Q AND NOT MM2VIS.bMsg1021 AND NOT MM2VIS.bMsg2101;
	xMsg3220.PT			:=	T#0s;
	xMsg3220.Prio		:=	4;
	xMsg3220.RiskClass	:=	4;
	xMsg3220.Reset		:=	FALSE;
	xMsg3220();
	MM2VIS.bMsg3220     := xMsg3220.Q;

	(* A3303 charge cooling water temperature high *)
	(*       temperature heat water return - low temp circuit *)
	xMsg3303.Enable		:=	FALSE;
	xMsg3303.Set 		:=	FALSE; 	(* actual not used *)
	xMsg3303.PT			:=	T#0s;
	xMsg3303.Prio		:=	3;
	xMsg3303.RiskClass	:=	4;
	xMsg3303.Reset		:=	FALSE;
	xMsg3303();
	MM2VIS.bMsg3303     := xMsg3303.Q;

	(* A3312 heat water return temperature after dump radiator signal failure trip (W3508)*)
	xMsg3312.Enable		:=	Para.bT_HW_ReAfEC_Active AND Para.bT_HW_ReAfEC_SF_Trip;
	xMsg3312.Set 		:=  NOT IN_HC.tT_HW_ReAfEC.GoodQual;
	xMsg3312.PT			:=	T#0s;
	xMsg3312.Prio		:=	3;
	xMsg3312.RiskClass	:=	4;
	xMsg3312.Reset		:=	FALSE;
	xMsg3312();
	MM2VIS.bMsg3312     := xMsg3312.Q;

	(* A3321 heat water return temperature before engine signal failure (W3526)*)
	xMsg3321.Enable		:=	Para.bT_HW_ReBeEng_Active AND Para.bT_HW_ReBeEng_SF_Trip;
	xMsg3321.Set 		:=  NOT IN_HC.tT_HW_ReBeEng.GoodQual;
	xMsg3321.PT			:=	T#0s;
	xMsg3321.Prio		:=	3;
	xMsg3321.RiskClass	:=	4;
	xMsg3321.Reset		:=	FALSE;
	xMsg3321();
	MM2VIS.bMsg3321     := xMsg3321.Q;

	(* W3402 engine cooling water pressure low *)
	xMsg3402.Enable		:=	TRUE;
	xMsg3402.Set		:=	(bPr_ECW_LimOp AND IN_HC.tT_ECW.Ai > 80.0) OR bPr_ECW_Lo AND NOT MM2VIS.bMsg1019;
	xMsg3402.PT			:=	T#0s;
	xMsg3402.Prio		:=	4;
	xMsg3402.RiskClass	:=	4;
	xMsg3402.Reset		:=	FALSE;
	xMsg3402();
	MM2VIS.bMsg3402     := xMsg3402.Q;

	(* W3404 water pressure cooler circuit low *)
	xMsg3404.Enable		:=	TRUE;
	xMsg3404.Set		:=	NOT IN_HC.tPr_CCircuit_Lo.Di;
	xMsg3404.PT			:=	T#10s;
	xMsg3404.Prio		:=	4;
	xMsg3404.RiskClass	:=	4;
	xMsg3404.Reset		:=	FALSE;
	xMsg3404();
	MM2VIS.bMsg3404     := xMsg3404.Q;
	OUT_HC.bMsg3404		:= xMsg3404.Q;

	(* W3406 engine cooling water pressure high *)
	xTP_3406(IN:= bN_EngStart, PT:= T#20s);

	xMsg3406.Enable		:=	TRUE;
	xMsg3406.Set 		:=  bPr_ECW_Hi AND NOT xTP_3406.Q;
	xMsg3406.PT			:=	T#0s;
	xMsg3406.Prio		:=	4;
	xMsg3406.RiskClass	:=	4;
	xMsg3406.Reset		:=	FALSE;
	xMsg3406();
	MM2VIS.bMsg3406     := xMsg3406.Q;

	(* W3407 outdoor temperature measuring signal failure *)
	xMsg3407.Enable		:=	Para.bT_AirOutdoor_Active AND IN_HC.tPB2MM.bParaSetupOk;
	xMsg3407.Set		:=	NOT IN_HC.tT_AirOutdoor.GoodQual;
	xMsg3407.PT			:=	T#0s;
	xMsg3407.Prio		:=	4;
	xMsg3407.RiskClass	:=	4;
	xMsg3407.Reset		:=	FALSE;
	xMsg3407();
	MM2VIS.bMsg3407		:=	xMsg3407.Q;

	(* W3492 temperature engine cooling water before charge cooler signal failure  *)
	xMsg3492.Enable		:=	Para.bT_ECW_bChC_HT_Active;
	xMsg3492.Set		:=	IN_HC.tPB2MM.bParaSetupOk AND NOT IN_HC.tT_ECW_bChC_HT.GoodQual;
	xMsg3492.PT			:=	T#0s;
	xMsg3492.Prio		:=	4;
	xMsg3492.RiskClass	:=	4;
	xMsg3492.Reset		:=	FALSE;
	xMsg3492();
	MM2VIS.bMsg3492		:=	xMsg3492.Q;

	(* W3493 temperature engine cooling water before oil cooler signal failure *)
	xMsg3493.Enable		:=	Para.bT_ECW_bOilC_Active;
	xMsg3493.Set		:=	IN_HC.tPB2MM.bParaSetupOk AND NOT IN_HC.tT_ECW_bOilC.GoodQual;
	xMsg3493.PT			:=	T#0s;
	xMsg3493.Prio		:=	4;
	xMsg3493.RiskClass	:=	4;
	xMsg3493.Reset		:=	FALSE;
	xMsg3493();
	MM2VIS.bMsg3493		:=	xMsg3493.Q;

	(* W3494 temperature engine cooling water before engine cooling water cooler signal failure  *)
	xMsg3494.Enable		:=	Para.bT_ECW_bECWC_Active;
	xMsg3494.Set		:=	IN_HC.tPB2MM.bParaSetupOk AND NOT IN_HC.tT_ECW_bECWC.GoodQual;
	xMsg3494.PT			:=	T#0s;
	xMsg3494.Prio		:=	4;
	xMsg3494.RiskClass	:=	4;
	xMsg3494.Reset		:=	FALSE;
	xMsg3494();
	MM2VIS.bMsg3494		:=	xMsg3494.Q;

	(* W3508 heat water return temperature after dump radiator signal failure (A3312)*)
	xMsg3508.Enable		:=	Para.bT_HW_ReAfEC_Active AND NOT Para.bT_HW_ReAfEC_SF_Trip AND IN_HC.tPB2MM.bParaSetupOk;
	xMsg3508.Set 		:=  NOT IN_HC.tT_HW_ReAfEC.GoodQual;
	xMsg3508.PT			:=	T#0s;
	xMsg3508.Prio		:=	4;
	xMsg3508.RiskClass	:=	4;
	xMsg3508.Reset		:=	FALSE;
	xMsg3508();
	MM2VIS.bMsg3508     := xMsg3508.Q;

	(* W3509 heat water return temperature after dump radiator high *)
	xMsg3509.Enable		:=	Para.bT_HW_ReAfEC_Active;
	xMsg3509.Set 		:=	bT_HW_ReAfEC_Hi AND NOT MM2VIS.bMsg3508 AND NOT MM2VIS.bMsg3312;
	xMsg3509.PT			:=	T#0s;
	xMsg3509.Prio		:=	4;
	xMsg3509.RiskClass	:=	4;
	xMsg3509.Reset		:=	FALSE;
	xMsg3509();
	MM2VIS.bMsg3509     := xMsg3509.Q;

	(* W3521 charge cooling water temperature high *)
	xGRMAX_T_HW_Re_LT_Hi(In:= IN_HC.tT_HW_Re_LT.Ai, Gw:= Para.rT_HW_Re_LT_LimHi, Hy:= Para.rT_HW_Re_LT_HyHi);
	xTON_3521(IN:= (xGRMAX_T_HW_Re_LT_Hi.Q AND Para.bT_HW_Re_LT_Active AND NOT xMsg3590.Q) OR NOT IN_HC.tT_ChCW_Hi.Di, PT:= T#10s);

	xMsg3521.Enable		:=	TRUE;
	xMsg3521.Set 		:=  xTON_3521.Q AND xTON_EngRunAnd10s.Q;
	xMsg3521.PT			:=	T#0s;
	xMsg3521.Prio		:=	4;
	xMsg3521.RiskClass	:=	4;
	xMsg3521.Reset		:=	FALSE;
	xMsg3521();
	MM2VIS.bMsg3521     := xMsg3521.Q;

	(* W3526 heating water return temperature before engine signal failure (A3321)*)
	xMsg3526.Enable		:=	Para.bT_HW_ReBeEng_Active AND NOT Para.bT_HW_ReBeEng_SF_Trip AND IN_HC.tPB2MM.bParaSetupOk;
	xMsg3526.Set 		:=  NOT IN_HC.tT_HW_ReBeEng.GoodQual;
	xMsg3526.PT			:=	T#0s;
	xMsg3526.Prio		:=	4;
	xMsg3526.RiskClass	:=	4;
	xMsg3526.Reset		:=	FALSE;
	xMsg3526();
	MM2VIS.bMsg3526     := xMsg3526.Q;

	(* W3527 heating water return temperature before engine high *)
	xTON_3527(IN:= bT_HW_ReBeEng_Hi AND IN_HC.tT_HW_ReBeEng.GoodQual, PT:= T#10s);

	xMsg3527.Enable		:=	Para.bT_HW_ReBeEng_Active;
	xMsg3527.Set 		:=  xTON_EngRunAnd10s.Q AND xTON_3527.Q;
	xMsg3527.PT			:=	T#0s;
	xMsg3527.Prio		:=	4;
	xMsg3527.RiskClass	:=	4;
	xMsg3527.Reset		:=	FALSE;
	xMsg3527();
	MM2VIS.bMsg3527     := xMsg3527.Q;

	(* W3590 signal failure charge cooling water temperature - low temp circuit *)
	(*       temperature heat water return - low temp circuit *)
	xMsg3590.Enable		:=	Para.bT_HW_Re_LT_Active AND IN_HC.tPB2MM.bParaSetupOk;
	xMsg3590.Set 		:=  NOT IN_HC.tT_HW_Re_LT.GoodQual;
	xMsg3590.PT			:=	T#0s;
	xMsg3590.Prio		:=	4;
	xMsg3590.RiskClass	:=	4;
	xMsg3590.Reset		:=	FALSE;
	xMsg3590();
	MM2VIS.bMsg3590     := xMsg3590.Q;

	(* W9226 Charge cooler 2 water pressure low *)
	xMsg9226.Enable		:=	TRUE;
	xMsg9226.Set		:=	NOT IN_HC.tPr_ChC2_Lo.Di;
	xMsg9226.PT			:=	T#10s;
	xMsg9226.Prio		:=	4;
	xMsg9226.RiskClass	:=	4;
	xMsg9226.Reset		:=	FALSE;
	xMsg9226();
	MM2VIS.bMsg9226     := xMsg9226.Q;
	OUT_HC.bMsg9226     := xMsg9226.Q;

	(* W9228 Charge cooler 2 failure *)
	xTON_ChC2_FanRdy(IN:= (IN_HC.tAuxV_Supply_Ok.Di AND IN_HC.tAuxV_Aux_ok.Di) AND NOT IN_HC.tChC2_FanRdy.Di, PT:= T#10s);

	xMsg9228.Enable		:=	TRUE;
	xMsg9228.Set		:=	NOT bNoMon4BlackStart AND(xTON_ChC2_FanRdy.Q OR NOT IN_HC.tChC2_Failure.Di);
	xMsg9228.PT			:=	T#0s;
	xMsg9228.Prio		:=	4;
	xMsg9228.RiskClass	:=	4;
	xMsg9228.Reset		:=	FALSE;
	xMsg9228();
	MM2VIS.bMsg9228     := xMsg9228.Q;

	(* W9229 Charge cooler 2 water temperature high *)
	xGRMAX_T_ChC2_Re_LT_Hi(In:= IN_HC.tT_ChC2_Re_LT.Ai, Gw:= Para.rT_ChC2_Re_LT_LimHi, Hy:= Para.rT_ChC2_Re_LT_HyHi);
	xTON_9229(IN:= (xGRMAX_T_ChC2_Re_LT_Hi.Q AND Para.bT_ChC2_Re_LT_Active AND NOT xMsg9232.Q) OR NOT IN_HC.tT_ChC2W_Hi.Di, PT:= T#10s);

	xMsg9229.Enable		:=	TRUE;
	xMsg9229.Set 		:=  xTON_9229.Q AND xTON_EngRunAnd10s.Q;
	xMsg9229.PT			:=	T#0s;
	xMsg9229.Prio		:=	4;
	xMsg9229.RiskClass	:=	4;
	xMsg9229.Reset		:=	FALSE;
	xMsg9229();
	MM2VIS.bMsg9229     := xMsg9229.Q;

	(* W9230 Measuring signal failure position temperature-control-valve charge cooler 2 circuit *)
	xMsg9230.Enable		:=	Para.bPos_ChC2_Valve;
	xMsg9230.Set 		:= 	IN_HC.tPB2MM.bParaSetupOk AND NOT IN_HC.tPos_ChC2_Valve.GoodQual;
	xMsg9230.PT			:=	T#0s;
	xMsg9230.Prio		:=	4;
	xMsg9230.RiskClass	:=	4;
	xMsg9230.Reset		:=	FALSE;
	xMsg9230();
	MM2VIS.bMsg9230     := xMsg9230.Q;

	(* W9231 Measuring signal failure supply water temperature charge cooler 2 circuit *)
	xMsg9231.Enable		:=	Para.bT_ChC2_Su_LT_Active;
	xMsg9231.Set		:=	IN_HC.tPB2MM.bParaSetupOk AND NOT IN_HC.tT_ChC2_Su_LT.GoodQual;
	xMsg9231.PT			:=	T#0s;
	xMsg9231.Prio		:=	4;
	xMsg9231.RiskClass	:=	4;
	xMsg9231.Reset		:=	FALSE;
	xMsg9231();
	MM2VIS.bMsg9231     := xMsg9231.Q;

	(* W9232 Measuring signal failure return water temperature charge cooler 2 circuit *)
	(*       return temperature - 2nd low temp circuit *)
	xMsg9232.Enable		:=	Para.bT_ChC2_Re_LT_Active AND IN_HC.tPB2MM.bParaSetupOk;
	xMsg9232.Set 		:=  NOT IN_HC.tT_ChC2_Re_LT.GoodQual;
	xMsg9232.PT			:=	T#0s;
	xMsg9232.Prio		:=	4;
	xMsg9232.RiskClass	:=	4;
	xMsg9232.Reset		:=	FALSE;
	xMsg9232();
	MM2VIS.bMsg9232     := xMsg9232.Q;

	(* W9588 Heating water supply temperature unit maximum *)						(* SAFETY PLC *)
	xMsg9588.Enable	   	:= Para.bT_HW_Su_Unit_Active;
	xMsg9588.Set	  	:= IN_HC.tT_HW_Su_Unit.Ai > Para.rT_HW_Su_Unit_LimHi;
	xMsg9588.PT	       	:= T#0s;
	xMsg9588.Prio	   	:= 4;
	xMsg9588.RiskClass	:= 4;
	xMsg9588.Reset	   	:= FALSE;
	xMsg9588();
	MM2VIS.bMsg9588		:= xMsg9588.Q;

	(* W9589 Heating water supply temperature unit measuring signal failure *)		(* SAFETY PLC *)
	xMsg9589.Enable	   	:= Para.bT_HW_Su_Unit_Active;
	xMsg9589.Set	  	:= NOT IN_HC.tT_HW_Su_Unit.GoodQual;
	xMsg9589.PT	       	:= T#0s;
	xMsg9589.Prio	   	:= 4;
	xMsg9589.RiskClass	:= 4;
	xMsg9589.Reset	   	:= FALSE;
	xMsg9589();
	MM2VIS.bMsg9589		:= xMsg9589.Q;

	(*---------------------------------------------------------------------------*)
	(* operating messages > AMM *)
	(* B9098 Valve heating in operation *)
	xMsg9098.Enable		:=	bValHeater_Dem_Exist;
	xMsg9098.Set		:= 	OUT_HC.tValHeater_Dem.Do;
	xMsg9098.Reset		:=	TRUE;
	xMsg9098();
	MM2VIS.bMsg9098		:=	xMsg9098.Q;

	(* B9099 Ring heater for cooling fan in operation *)
	xMsg9099.Enable		:=	bFanRingHeater_Dem_Exist;
	xMsg9099.Set		:= 	OUT_HC.tFanRingHeater_Dem.Do;
	xMsg9099.Reset		:=	TRUE;
	xMsg9099();
	MM2VIS.bMsg9099		:=	xMsg9099.Q;

	(*---------------------------------------------------------------------------*)
	(* general alarms for further module operations *)
	bGnlTrip1   := OUT_HC.tHC2AB.bGnlTrip1   OR IN_HC.tAB2HC.bGnlTrip1;
	bGnlTrip2   := OUT_HC.tHC2AB.bGnlTrip2   OR IN_HC.tAB2HC.bGnlTrip2;
	bGnlTrip3   := OUT_HC.tHC2AB.bGnlTrip3   OR IN_HC.tAB2HC.bGnlTrip3;
	bGnlWarning := OUT_HC.tHC2AB.bGnlWarning OR IN_HC.tAB2HC.bGnlWarning;

	bGnlTrip    := bGnlTrip1 OR bGnlTrip2 OR bGnlTrip3;

(*******************************************************************************)
END_PROGRAM
```

#### MsgHCInit.st
```iecst
(*******************************************************************************
Msg_HC	 			 alarms generation heating cooling

This code is confidential and proprietary to the INNIO Company.
It may not be used in any form, or reproduced in any manner,
without written permission of the INNIO Company.
Copyright, INNIO Company, 2019

Customized modifications: -
------------------------

History:
-------
V0.00.0	29.07.2011	lettenb.	new

Instructions for use:
--------------------
1) declare alarm with function block "Msg"

2) use template to create a new alarm, substitue 0000 by message number:

	xMsg0000.Num		:=	0000;					alarm number
	xMsg0000.AmmSysAdr	:=  iAdrAmmBase2MM;			do not change
	xMsg0000.AmmOutAdr	:=  iAdrMM2AmmBase;			do not change

3) 	set alarm number

Outstandings:
------------

(*******************************************************************************)
PROGRAM _INIT

	iAdrAmmBase2MM		:=  ADR(IN_HC.tAB2HC);
	iAdrMM2AmmBase		:=  ADR(OUT_HC.tHC2AB);

	(*---------------------------------------------------------------------------*)

	xMsg1019.Num		:=	1019;
	xMsg1019.AmmInAdr	:=  iAdrAmmBase2MM;
	xMsg1019.AmmOutAdr	:=  iAdrMM2AmmBase;

	xMsg1021.Num		:=	1021;
	xMsg1021.AmmInAdr	:=  iAdrAmmBase2MM;
	xMsg1021.AmmOutAdr	:=  iAdrMM2AmmBase;

	xMsg1032.Num		:=	1032;
	xMsg1032.AmmInAdr	:=  iAdrAmmBase2MM;
	xMsg1032.AmmOutAdr	:=  iAdrMM2AmmBase;

	xMsg1033.Num		:=	1033;
	xMsg1033.AmmInAdr	:=  iAdrAmmBase2MM;
	xMsg1033.AmmOutAdr	:=  iAdrMM2AmmBase;

	xMsg1034.Num		:=	1034;
	xMsg1034.AmmInAdr	:=  iAdrAmmBase2MM;
	xMsg1034.AmmOutAdr	:=  iAdrMM2AmmBase;

	xMsg1035.Num		:=	1035;
	xMsg1035.AmmInAdr	:=  iAdrAmmBase2MM;
	xMsg1035.AmmOutAdr	:=  iAdrMM2AmmBase;

	xMsg1050.Num		:=	1050;
	xMsg1050.AmmInAdr	:=  iAdrAmmBase2MM;
	xMsg1050.AmmOutAdr	:=  iAdrMM2AmmBase;

	xMsg1063.Num		:=	1063;
	xMsg1063.AmmInAdr	:=  iAdrAmmBase2MM;
	xMsg1063.AmmOutAdr	:=  iAdrMM2AmmBase;

	xMsg1070.Num		:=	1070;
	xMsg1070.AmmInAdr	:=  iAdrAmmBase2MM;
	xMsg1070.AmmOutAdr	:=  iAdrMM2AmmBase;

	xMsg1071.Num		:=	1071;
	xMsg1071.AmmInAdr	:=  iAdrAmmBase2MM;
	xMsg1071.AmmOutAdr	:=  iAdrMM2AmmBase;

	xMsg1130.Num		:=	1130;
	xMsg1130.AmmInAdr	:=  iAdrAmmBase2MM;
	xMsg1130.AmmOutAdr	:=  iAdrMM2AmmBase;

	xMsg1145.Num		:=	1145;
	xMsg1145.AmmInAdr	:=  iAdrAmmBase2MM;
	xMsg1145.AmmOutAdr	:=  iAdrMM2AmmBase;

	xMsg1167.Num		:=	1167;
	xMsg1167.AmmInAdr	:=  iAdrAmmBase2MM;
	xMsg1167.AmmOutAdr	:=  iAdrMM2AmmBase;

	xMsg1186.Num		:=	1186;
	xMsg1186.AmmInAdr	:=  iAdrAmmBase2MM;
	xMsg1186.AmmOutAdr	:=  iAdrMM2AmmBase;

	xMsg1187.Num		:=	1187;
	xMsg1187.AmmInAdr	:=  iAdrAmmBase2MM;
	xMsg1187.AmmOutAdr	:=  iAdrMM2AmmBase;

	xMsg2101.Num		:=	2101;
	xMsg2101.AmmInAdr	:=  iAdrAmmBase2MM;
	xMsg2101.AmmOutAdr	:=  iAdrMM2AmmBase;

	xMsg2104.Num		:=	2104;
	xMsg2104.AmmInAdr	:=  iAdrAmmBase2MM;
	xMsg2104.AmmOutAdr	:=  iAdrMM2AmmBase;

	xMsg2116.Num		:=	2116;
	xMsg2116.AmmInAdr	:=  iAdrAmmBase2MM;
	xMsg2116.AmmOutAdr	:=  iAdrMM2AmmBase;

	xMsg2117.Num		:=	2117;
	xMsg2117.AmmInAdr	:=  iAdrAmmBase2MM;
	xMsg2117.AmmOutAdr	:=  iAdrMM2AmmBase;

	xMsg2119.Num		:=	2119;
	xMsg2119.AmmInAdr	:=  iAdrAmmBase2MM;
	xMsg2119.AmmOutAdr	:=  iAdrMM2AmmBase;

	xMsg2341.Num		:=	2341;
	xMsg2341.AmmInAdr	:=  iAdrAmmBase2MM;
	xMsg2341.AmmOutAdr	:=  iAdrMM2AmmBase;

	xMsg2342.Num		:=	2342;
	xMsg2342.AmmInAdr	:=  iAdrAmmBase2MM;
	xMsg2342.AmmOutAdr	:=  iAdrMM2AmmBase;

	xMsg2343.Num		:=	2343;
	xMsg2343.AmmInAdr	:=  iAdrAmmBase2MM;
	xMsg2343.AmmOutAdr	:=  iAdrMM2AmmBase;

	xMsg2428.Num		:=	2428;//SWAT920/1
	xMsg2428.AmmInAdr	:=  iAdrAmmBase2MM;
	xMsg2428.AmmOutAdr	:=  iAdrMM2AmmBase;

	xMsg2429.Num		:=	2429;//SWAT920/1
	xMsg2429.AmmInAdr	:=  iAdrAmmBase2MM;
	xMsg2429.AmmOutAdr	:=  iAdrMM2AmmBase;

	xMsg2430.Num		:=	2430;//SWAT920/1
	xMsg2430.AmmInAdr	:=  iAdrAmmBase2MM;
	xMsg2430.AmmOutAdr	:=  iAdrMM2AmmBase;

	xMsg2638.Num		:=	2638;
	xMsg2638.AmmInAdr	:=  iAdrAmmBase2MM;
	xMsg2638.AmmOutAdr	:=  iAdrMM2AmmBase;

	xMsg2639.Num		:=	2639;
	xMsg2639.AmmInAdr	:=  iAdrAmmBase2MM;
	xMsg2639.AmmOutAdr	:=  iAdrMM2AmmBase;

	xMsg2640.Num		:=	2640;
	xMsg2640.AmmInAdr	:=  iAdrAmmBase2MM;
	xMsg2640.AmmOutAdr	:=  iAdrMM2AmmBase;

	xMsg2641.Num		:=	2641;
	xMsg2641.AmmInAdr	:=  iAdrAmmBase2MM;
	xMsg2641.AmmOutAdr	:=  iAdrMM2AmmBase;

	xMsg2647.Num 		:= 	2647;
	xMsg2647.AmmInAdr 	:=  iAdrAmmBase2MM;
	xMsg2647.AmmOutAdr 	:=  iAdrMM2AmmBase;

	xMsg2667.Num 		:= 	2667;
	xMsg2667.AmmInAdr 	:=  iAdrAmmBase2MM;
	xMsg2667.AmmOutAdr 	:=  iAdrMM2AmmBase;

	xMsg2675.Num 		:= 	2675;
	xMsg2675.AmmInAdr 	:=  iAdrAmmBase2MM;
	xMsg2675.AmmOutAdr 	:=  iAdrMM2AmmBase;

	xMsg2676.Num 		:= 	2676;
	xMsg2676.AmmInAdr 	:=  iAdrAmmBase2MM;
	xMsg2676.AmmOutAdr 	:=  iAdrMM2AmmBase;

	xMsg2677.Num 		:= 	2677;
	xMsg2677.AmmInAdr 	:=  iAdrAmmBase2MM;
	xMsg2677.AmmOutAdr 	:=  iAdrMM2AmmBase;

	xMsg2678.Num 		:= 	2678;
	xMsg2678.AmmInAdr 	:=  iAdrAmmBase2MM;
	xMsg2678.AmmOutAdr 	:=  iAdrMM2AmmBase;

	xMsg2679.Num 		:= 	2679;
	xMsg2679.AmmInAdr 	:=  iAdrAmmBase2MM;
	xMsg2679.AmmOutAdr 	:=  iAdrMM2AmmBase;

	xMsg2680.Num 		:= 	2680;
	xMsg2680.AmmInAdr 	:=  iAdrAmmBase2MM;
	xMsg2680.AmmOutAdr 	:=  iAdrMM2AmmBase;

	xMsg2681.Num 		:= 	2681;
	xMsg2681.AmmInAdr 	:=  iAdrAmmBase2MM;
	xMsg2681.AmmOutAdr 	:=  iAdrMM2AmmBase;

	xMsg2682.Num 		:= 	2682;
	xMsg2682.AmmInAdr 	:=  iAdrAmmBase2MM;
	xMsg2682.AmmOutAdr 	:=  iAdrMM2AmmBase;

	xMsg2683.Num 		:= 	2683;
	xMsg2683.AmmInAdr 	:=  iAdrAmmBase2MM;
	xMsg2683.AmmOutAdr 	:=  iAdrMM2AmmBase;

	xMsg2684.Num 		:= 	2684;
	xMsg2684.AmmInAdr 	:=  iAdrAmmBase2MM;
	xMsg2684.AmmOutAdr 	:=  iAdrMM2AmmBase;

	xMsg2685.Num 		:= 	2685;
	xMsg2685.AmmInAdr 	:=  iAdrAmmBase2MM;
	xMsg2685.AmmOutAdr 	:=  iAdrMM2AmmBase;

	xMsg2686.Num 		:= 	2686;
	xMsg2686.AmmInAdr 	:=  iAdrAmmBase2MM;
	xMsg2686.AmmOutAdr 	:=  iAdrMM2AmmBase;

	xMsg2687.Num 		:= 	2687;
	xMsg2687.AmmInAdr 	:=  iAdrAmmBase2MM;
	xMsg2687.AmmOutAdr 	:=  iAdrMM2AmmBase;

	xMsg2710.Num 		:= 	2710;
	xMsg2710.AmmInAdr 	:=  iAdrAmmBase2MM;
	xMsg2710.AmmOutAdr 	:=  iAdrMM2AmmBase;

	xMsg2711.Num 		:= 	2711;
	xMsg2711.AmmInAdr 	:=  iAdrAmmBase2MM;
	xMsg2711.AmmOutAdr 	:=  iAdrMM2AmmBase;

	xMsg2712.Num 		:= 	2712;
	xMsg2712.AmmInAdr 	:=  iAdrAmmBase2MM;
	xMsg2712.AmmOutAdr 	:=  iAdrMM2AmmBase;

	xMsg2713.Num 		:= 	2713;
	xMsg2713.AmmInAdr 	:=  iAdrAmmBase2MM;
	xMsg2713.AmmOutAdr 	:=  iAdrMM2AmmBase;

	xMsg2714.Num 		:= 	2714;
	xMsg2714.AmmInAdr 	:=  iAdrAmmBase2MM;
	xMsg2714.AmmOutAdr 	:=  iAdrMM2AmmBase;

	xMsg2715.Num 		:= 	2715;
	xMsg2715.AmmInAdr 	:=  iAdrAmmBase2MM;
	xMsg2715.AmmOutAdr 	:=  iAdrMM2AmmBase;

	xMsg2716.Num 		:= 	2716;
	xMsg2716.AmmInAdr 	:=  iAdrAmmBase2MM;
	xMsg2716.AmmOutAdr 	:=  iAdrMM2AmmBase;

	xMsg2717.Num 		:= 	2717;
	xMsg2717.AmmInAdr 	:=  iAdrAmmBase2MM;
	xMsg2717.AmmOutAdr 	:=  iAdrMM2AmmBase;

	xMsg2718.Num 		:= 	2718;
	xMsg2718.AmmInAdr 	:=  iAdrAmmBase2MM;
	xMsg2718.AmmOutAdr 	:=  iAdrMM2AmmBase;

	xMsg2719.Num 		:= 	2719;
	xMsg2719.AmmInAdr 	:=  iAdrAmmBase2MM;
	xMsg2719.AmmOutAdr 	:=  iAdrMM2AmmBase;

	xMsg2720.Num 		:= 	2720;
	xMsg2720.AmmInAdr 	:=  iAdrAmmBase2MM;
	xMsg2720.AmmOutAdr 	:=  iAdrMM2AmmBase;

	xMsg2721.Num 		:= 	2721;
	xMsg2721.AmmInAdr 	:=  iAdrAmmBase2MM;
	xMsg2721.AmmOutAdr 	:=  iAdrMM2AmmBase;

	xMsg2731.Num 		:= 	2731;
	xMsg2731.AmmInAdr 	:=  iAdrAmmBase2MM;
	xMsg2731.AmmOutAdr 	:=  iAdrMM2AmmBase;

	xMsg2732.Num 		:= 	2732;
	xMsg2732.AmmInAdr 	:=  iAdrAmmBase2MM;
	xMsg2732.AmmOutAdr 	:=  iAdrMM2AmmBase;

	xMsg2733.Num 		:= 	2733;
	xMsg2733.AmmInAdr 	:=  iAdrAmmBase2MM;
	xMsg2733.AmmOutAdr 	:=  iAdrMM2AmmBase;

	xMsg2734.Num 		:= 	2734;
	xMsg2734.AmmInAdr 	:=  iAdrAmmBase2MM;
	xMsg2734.AmmOutAdr 	:=  iAdrMM2AmmBase;

	xMsg2735.Num 		:= 	2735;
	xMsg2735.AmmInAdr 	:=  iAdrAmmBase2MM;
	xMsg2735.AmmOutAdr 	:=  iAdrMM2AmmBase;

	xMsg2736.Num 		:= 	2736;
	xMsg2736.AmmInAdr 	:=  iAdrAmmBase2MM;
	xMsg2736.AmmOutAdr 	:=  iAdrMM2AmmBase;

	xMsg2750.Num 		:= 	2750;
	xMsg2750.AmmInAdr 	:=  iAdrAmmBase2MM;
	xMsg2750.AmmOutAdr 	:=  iAdrMM2AmmBase;

	xMsg2751.Num 		:= 	2751;
	xMsg2751.AmmInAdr 	:=  iAdrAmmBase2MM;
	xMsg2751.AmmOutAdr 	:=  iAdrMM2AmmBase;

	xMsg2752.Num 		:= 	2752;
	xMsg2752.AmmInAdr 	:=  iAdrAmmBase2MM;
	xMsg2752.AmmOutAdr 	:=  iAdrMM2AmmBase;

	xMsg2763.Num 		:= 	2763;
	xMsg2763.AmmInAdr 	:=  iAdrAmmBase2MM;
	xMsg2763.AmmOutAdr 	:=  iAdrMM2AmmBase;

	xMsg3220.Num		:=	3220;
	xMsg3220.AmmInAdr	:=  iAdrAmmBase2MM;
	xMsg3220.AmmOutAdr	:=  iAdrMM2AmmBase;

	xMsg3303.Num		:=	3303;
	xMsg3303.AmmInAdr	:=  iAdrAmmBase2MM;
	xMsg3303.AmmOutAdr	:=  iAdrMM2AmmBase;

	xMsg3312.Num		:=	3312;
	xMsg3312.AmmInAdr	:=  iAdrAmmBase2MM;
	xMsg3312.AmmOutAdr	:=  iAdrMM2AmmBase;

	xMsg3321.Num		:=	3321;
	xMsg3321.AmmInAdr	:=  iAdrAmmBase2MM;
	xMsg3321.AmmOutAdr	:=  iAdrMM2AmmBase;

	xMsg3402.Num		:=	3402;
	xMsg3402.AmmInAdr	:=  iAdrAmmBase2MM;
	xMsg3402.AmmOutAdr	:=  iAdrMM2AmmBase;

	xMsg3404.Num		:=	3404;
	xMsg3404.AmmInAdr	:=  iAdrAmmBase2MM;
	xMsg3404.AmmOutAdr	:=  iAdrMM2AmmBase;

	xMsg3406.Num		:=	3406;
	xMsg3406.AmmInAdr	:=  iAdrAmmBase2MM;
	xMsg3406.AmmOutAdr	:=  iAdrMM2AmmBase;

	xMsg3407.Num		:=	3407;
    xMsg3407.AmmInAdr	:=  iAdrAmmBase2MM;
	xMsg3407.AmmOutAdr	:=  iAdrMM2AmmBase;

	xMsg3492.Num		:=	3492;
    xMsg3492.AmmInAdr	:=  iAdrAmmBase2MM;
	xMsg3492.AmmOutAdr	:=  iAdrMM2AmmBase;

	xMsg3493.Num		:=	3493;
    xMsg3493.AmmInAdr	:=  iAdrAmmBase2MM;
	xMsg3493.AmmOutAdr	:=  iAdrMM2AmmBase;

	xMsg3494.Num		:=	3494;
    xMsg3494.AmmInAdr	:=  iAdrAmmBase2MM;
	xMsg3494.AmmOutAdr	:=  iAdrMM2AmmBase;

	xMsg3508.Num		:=	3508;
	xMsg3508.AmmInAdr	:=  iAdrAmmBase2MM;
	xMsg3508.AmmOutAdr	:=  iAdrMM2AmmBase;

	xMsg3509.Num		:=	3509;
	xMsg3509.AmmInAdr	:=  iAdrAmmBase2MM;
	xMsg3509.AmmOutAdr	:=  iAdrMM2AmmBase;

	xMsg3521.Num		:=	3521;
	xMsg3521.AmmInAdr	:=  iAdrAmmBase2MM;
	xMsg3521.AmmOutAdr	:=  iAdrMM2AmmBase;

	xMsg3526.Num		:=	3526;
	xMsg3526.AmmInAdr	:=  iAdrAmmBase2MM;
	xMsg3526.AmmOutAdr	:=  iAdrMM2AmmBase;

	xMsg3527.Num		:=	3527;
	xMsg3527.AmmInAdr	:=  iAdrAmmBase2MM;
	xMsg3527.AmmOutAdr	:=  iAdrMM2AmmBase;

	xMsg3590.Num		:=	3590;
	xMsg3590.AmmInAdr	:=  iAdrAmmBase2MM;
	xMsg3590.AmmOutAdr	:=  iAdrMM2AmmBase;

	xMsg9226.Num		:=	9226;
	xMsg9226.AmmInAdr	:=  iAdrAmmBase2MM;
	xMsg9226.AmmOutAdr	:=  iAdrMM2AmmBase;

	xMsg9098.Num		:=	9098;
	xMsg9098.AmmInAdr	:=  iAdrAmmBase2MM;
	xMsg9098.AmmOutAdr	:=  iAdrMM2AmmBase;

	xMsg9099.Num		:=	9099;
	xMsg9099.AmmInAdr	:=  iAdrAmmBase2MM;
	xMsg9099.AmmOutAdr	:=  iAdrMM2AmmBase;

	xMsg9228.Num		:=	9228;
	xMsg9228.AmmInAdr	:=  iAdrAmmBase2MM;
	xMsg9228.AmmOutAdr	:=  iAdrMM2AmmBase;

	xMsg9229.Num		:=	9229;
	xMsg9229.AmmInAdr	:=  iAdrAmmBase2MM;
	xMsg9229.AmmOutAdr	:=  iAdrMM2AmmBase;

	xMsg9230.Num		:=	9230;
	xMsg9230.AmmInAdr	:=  iAdrAmmBase2MM;
	xMsg9230.AmmOutAdr	:=  iAdrMM2AmmBase;

	xMsg9231.Num		:=	9231;
	xMsg9231.AmmInAdr	:=  iAdrAmmBase2MM;
	xMsg9231.AmmOutAdr	:=  iAdrMM2AmmBase;

	xMsg9232.Num		:=	9232;
	xMsg9232.AmmInAdr	:=  iAdrAmmBase2MM;
	xMsg9232.AmmOutAdr	:=  iAdrMM2AmmBase;

	xMsg9588.Num		:= 9588;
	xMsg9588.AmmInAdr	:= iAdrAmmBase2MM;
	xMsg9588.AmmOutAdr	:= iAdrMM2AmmBase;

	xMsg9589.Num		:= 9589;
	xMsg9589.AmmInAdr	:= iAdrAmmBase2MM;
	xMsg9589.AmmOutAdr	:= iAdrMM2AmmBase;
END_PROGRAM
```

#### MsgHC.var
```iecst
VAR
	bNoMon4BlackStart : BOOL; (*temporary no monitoring for engine blackstart *)
	iAdrAmmBase2MM : UDINT;
	iAdrMM2AmmBase : UDINT;
	xGRMAX_T_HW_Re_LT_Hi : GR_MAXR;
	xGRMAX_T_Su_PriCirc : GR_MAXR;
	xGRMAX_T_Re_PriCirc : GR_MAXR;
	xGRMAX_T_Su_SecCirc : GR_MAXR;
	xGRMAX_T_Re_SecCirc : GR_MAXR;
	xMsg1019 : Msg;
	xMsg1021 : Msg;
	xMsg1032 : Msg;
	xMsg1033 : Msg;
	xMsg1034 : Msg;
	xMsg1035 : Msg;
	xMsg1050 : Msg;
	xMsg1063 : Msg;
	xMsg1070 : Msg;
	xMsg1071 : Msg;
	xMsg1130 : Msg;
	xMsg1145 : Msg;
	xMsg1167 : Msg;
	xMsg1186 : Msg;
	xMsg1187 : Msg;
	xMsg2101 : Msg;
	xMsg2104 : Msg;
	xMsg2116 : Msg;
	xMsg2117 : Msg;
	xMsg2119 : Msg;
	xMsg2341 : Msg;
	xMsg2342 : Msg;
	xMsg2343 : Msg;
	xMsg2428 : Msg; (*SWAT920/1*)
	xMsg2429 : Msg; (*SWAT920/1*)
	xMsg2430 : Msg; (*SWAT920/1*)
	xMsg2638 : Msg;
	xMsg2639 : Msg;
	xMsg2640 : Msg;
	xMsg2641 : Msg;
	xMsg2647 : Msg;
	xMsg2667 : Msg;
	xMsg2675 : Msg;
	xMsg2676 : Msg;
	xMsg2677 : Msg;
	xMsg2678 : Msg;
	xMsg2679 : Msg;
	xMsg2680 : Msg;
	xMsg2681 : Msg;
	xMsg2682 : Msg;
	xMsg2683 : Msg;
	xMsg2684 : Msg;
	xMsg2685 : Msg;
	xMsg2686 : Msg;
	xMsg2687 : Msg;
	xMsg2710 : Msg;
	xMsg2711 : Msg;
	xMsg2712 : Msg;
	xMsg2713 : Msg;
	xMsg2714 : Msg;
	xMsg2715 : Msg;
	xMsg2716 : Msg;
	xMsg2717 : Msg;
	xMsg2718 : Msg;
	xMsg2719 : Msg;
	xMsg2720 : Msg;
	xMsg2721 : Msg;
	xMsg2736 : Msg;
	xMsg2731 : Msg;
	xMsg2732 : Msg;
	xMsg2733 : Msg;
	xMsg2734 : Msg;
	xMsg2735 : Msg;
	xMsg2750 : Msg;
	xMsg2751 : Msg;
	xMsg2752 : Msg;
	xMsg2763 : Msg;
	xMsg3220 : Msg;
	xMsg3303 : Msg;
	xMsg3312 : Msg;
	xMsg3321 : Msg;
	xMsg3402 : Msg;
	xMsg3404 : Msg;
	xMsg3406 : Msg;
	xMsg3407 : Msg;
	xMsg3492 : Msg;
	xMsg3493 : Msg;
	xMsg3494 : Msg;
	xMsg3508 : Msg;
	xMsg3509 : Msg;
	xMsg3521 : Msg;
	xMsg3526 : Msg;
	xMsg3527 : Msg;
	xMsg3590 : Msg;
	xMsg9098 : Msg;
	xMsg9099 : Msg;
	xMsg9226 : Msg;
	xMsg9228 : Msg;
	xMsg9229 : Msg;
	xMsg9230 : Msg;
	xMsg9231 : Msg;
	xMsg9232 : Msg;
	xMsg9588 : Msg; (*FuB*) (*SAFETY PLC*)
	xMsg9589 : Msg; (*FuB*) (*SAFETY PLC*)
	xTOF_EngDemEPS : TOF;
	xTON_1021 : TON;
	xTON_1167 : TON;
	xTON_3521 : TON;
	xTON_3527 : TON;
	xTON_ChC_FanRdy : TON;
	xTON_EngRunAnd10s : TON;
	xTON_EngRunAnd60s : TON;
	xTP_1019 : TP;
	xTP_1050 : TP;
	xTP_2104 : TP;
	xTP_3406 : TP;
	xTOF_CDP_Fail : TOF;
	xTON_CDP_Fail : TON;
	HBT_1 : BOOL;
	KTMA_VISA : BOOL;
	xTON_ChC2_FanRdy : TON;
	xGRMAX_T_ChC2_Re_LT_Hi : GR_MAXR;
	xTON_9229 : TON;
END_VAR
```

### Program Logical/HeatingCooling/vis_HC (IEC) - visualization

#### vis_HCCyclic.st
```iecst
(*******************************************************************************
vis			visualization

This code is confidential and proprietary to the INNIO Company.
It may not be used in any form, or reproduced in any manner,
without the express written permission of the INNIO Company.
Copyright, INNIO Company, 2025

Customized modifications: -
------------------------

History:
-------
V3.40.0	21.02.2013	lettenb.	tT_HW_Re_LT added
V3.99.0	24.04.2012	lettenb.	new
		25.09.2012				bEC_Dem added for diane_vis
V4.00.0 15.12.2014				tT_HW_Re_LT --> rT_HW_Re_LT, bugfix
								tPr_ECWaEng,tT_ECWbEng added
V4.03.0 06.07.2015				920 ECW + EO module signals added(TCA redesign)
        29.07.2015	plattner	heat circuit temperature added
        05.08.2015  Stary       primary/secondary temperatures added
 		07.08.2015  Denk		Manual operating auxiliaries control functionality added
V4.04.0 04.05.2016	lettenb.	rT_ECW_bChC_HT, rT_ECW_bOilC, rT_ECW_bECWC added
		21.10.2016				MM2VIS.bEC_On,MM2VIS.bChC_On added(stary)
V4.07.0	09.08.2018	Schmid		2nd low temperature charge cooling circuit added
V4.14.0 08.11.2024	Bacci		MM2VIS.bECW_ShutOffVal_Dem (exist), MM2VIS.bValHeater_Dem (exist), MM2VIS.bFanRingHeater_Dem (exist) added
V4.25.0	10.07.2025	Tinello		SafetyPLC: Added heating water supply temperature unit

Instructions for use:
--------------------
Outstandings:
------------
*******************************************************************************)
PROGRAM _CYCLIC

	MM2VIS.rT_AirOutdoor	:=	IN_HC.tT_AirOutdoor.Ai;
	MM2VIS.bECW_DemBpP		:=	bECW_DemBpP;
	MM2VIS.bEC_Stage1		:=	K_ST1 OR K_ST1_ManAuxCtr;
	MM2VIS.bEC_Stage2		:=	K_ST2 OR K_ST2_ManAuxCtr;
	MM2VIS.bEC_Dem			:=	K_ST1 OR K_ST2 OR K_ST1_ManAuxCtr OR K_ST2_ManAuxCtr;
	MM2VIS.iSumChC_Stages	:=	iSumChC_Stages;
	MM2VIS.iSumEC_Stages	:=	iSumEC_Stages;

	MM2VIS.rT_HW_ReBeEng	:=	IN_HC.tT_HW_ReBeEng.Ai;
	MM2VIS.rT_HW_ReAfEC		:=	IN_HC.tT_HW_ReAfEC.Ai;
	MM2VIS.rT_HW_Re			:=	IN_HC.tT_HW_Re.Ai;
	MM2VIS.rT_HW_Su			:=	IN_HC.tT_HW_Su.Ai;
	MM2VIS.rPr_ECW			:=	IN_HC.tPr_ECW.Ai;
	MM2VIS.rPr_ECWaEng		:=	IN_HC.tPr_ECWaEng.Ai;
	MM2VIS.rT_ECW			:=	IN_HC.tT_ECW.Ai;
	MM2VIS.rP_Red_T_HWR_Norm:=	OUT_HC.rP_Red_T_HWR_Norm;
	MM2VIS.rP_Red_T_ECW_Norm:=	OUT_HC.rP_Red_T_ECW_Norm;
	MM2VIS.rT_HW_Su_LT		:=	IN_HC.tT_HW_Su_LT.Ai;
	MM2VIS.rT_HW_Re_LT		:=	IN_HC.tT_HW_Re_LT.Ai;
	MM2VIS.rT_Su_PriCirc    :=  IN_HC.tT_Su_PriCirc.Ai;
	MM2VIS.rT_Re_PriCirc    :=  IN_HC.tT_Re_PriCirc.Ai;
	MM2VIS.rT_Su_SecCirc    :=  IN_HC.tT_Su_SecCirc.Ai;
	MM2VIS.rT_Re_SecCirc    :=  IN_HC.tT_Re_SecCirc.Ai;
	MM2VIS.rP_Heat          :=  IN_HC.tP_Heat.Ai;

	MM2VIS.rT_ECWbEng		:=	IN_HC.tT_ECWbEng.Ai;
	MM2VIS.rT_ECW_AfEng		:=	IN_HC.tT_ECW_AfEng.Ai;

	MM2VIS.rPr_HW_Su_LT		:=	IN_HC.tPr_HW_Su_LT.Ai;
	MM2VIS.rPr_HW_Su_HT		:=	IN_HC.tPr_HW_Su_HT.Ai;

	MM2VIS.rPr_HW_Re_LT         := IN_HC.tPr_HW_Re_LT.Ai;      (*pressure heat water return low temp.circuit M.07-PI-002*)
	MM2VIS.rPr_HW_Re_HT         := IN_HC.tPr_HW_Re_HT.Ai;      (*pressure heat water return high temp.circuit M.06-PI-002*)
	MM2VIS.rPr_HW_Re_PreH_ECW   := IN_HC.tPr_HW_Re_PreH_ECW.Ai;(*pressure heat water return preheating engine cooling water M.04-PI-005*)
	MM2VIS.rPr_HW_Re_PreH_EO    := IN_HC.tPr_HW_Re_PreH_EO.Ai; (*pressure heat water return preheating engine oil M.03-PI-005*)
	MM2VIS.rPr_EO_Mod_Out       := IN_HC.tPr_EO_Mod_Out.Ai;    (*pressure engine oil module outlet M.03-PI-006*) (*OldName:newPv; Cycle:5;*)
	MM2VIS.rT_ECW_Mod_In        := IN_HC.tT_ECW_Mod_In.Ai;     (*temperature engine cooling water, engine cooling water module inlet M.04-TI-003*)
	MM2VIS.rT_ECW_Mod_Out       := IN_HC.tT_ECW_Mod_Out.Ai;    (*temperature engine cooling water, engine cooling water module outlet M.04-TI-004*)
	MM2VIS.rT_EO_Mod_In         := IN_HC.tT_EO_Mod_In.Ai;      (*temperature engine oil, oil module inlet M.03-TI-004*)
	MM2VIS.rT_EO_Mod_Out        := IN_HC.tT_EO_Mod_Out.Ai;     (*temperature engine oil, oil module outlet M.03-TI-003*)
	MM2VIS.rT_HW_Su_PreH_ECW    := IN_HC.tT_HW_Su_PreH_ECW.Ai; (*temperature heat water supply preheating engine cooling water M.04-TI-005*)
	MM2VIS.rT_HW_Re_PreH_ECW    := IN_HC.tT_HW_Re_PreH_ECW.Ai; (*temperature heat water return preheating engine cooling water M.04-TI-006*)
	MM2VIS.rT_HW_Su_PreH_EO     := IN_HC.tT_HW_Su_PreH_EO.Ai;  (*temperature heat water supply preheating engine oil M.03-TI-005*)
	MM2VIS.rT_HW_Re_PreH_EO     := IN_HC.tT_HW_Re_PreH_EO.Ai;  (*temperature heat water return preheating engine oil M.03-TI-006*)
	MM2VIS.rT_ECW_bChC_HT     	:= IN_HC.tT_ECW_bChC_HT.Ai;	   (*temperature engine cooling water high temp.circ.before charge cooler M.06-TI-014*)
	MM2VIS.rT_ECW_bOilC     	:= IN_HC.tT_ECW_bOilC.Ai;	   (*temperature engine cooling water before oil cooler M.06-TI-020*)
	MM2VIS.rT_ECW_bECWC     	:= IN_HC.tT_ECW_bECWC.Ai;	   (*temperature engine cooling water before engine cooling water cooler M.06-TI-030*)

	MM2VIS.bEC_DemPump			:= OUT_HC.tEC_DemPump.Do;
	MM2VIS.bChC_DemPump			:= OUT_HC.tChC_DemPump.Do;
	MM2VIS.bEC_On     			:= (MM2VIS.iSumEC_Stages = 1  AND NOT MM2VIS.bMsg2116) OR (MM2VIS.iSumEC_Stages > 1  AND MM2VIS.bMsg2116);
	MM2VIS.bChC_On    			:= (MM2VIS.iSumChC_Stages = 1 AND NOT MM2VIS.bMsg2119) OR (MM2VIS.iSumChC_Stages > 1 AND MM2VIS.bMsg2119);

	MM2VIS.rT_CD_Su					:=	IN_HC.tT_CD_Su.Ai;
	MM2VIS.rT_CD_Re					:=	IN_HC.tT_CD_Re.Ai;
	MM2VIS.bBHV_Dem					:=	OUT_HC.tBHV_Dem.Do AND NOT MM2VIS.bMsg2736;
	MM2VIS.bCDP_Dem					:=	IN_HC.tCDP_Dem.Do AND NOT MM2VIS.bMsg2735;
	MM2VIS.rT_HW_HC_Re				:=	IN_HC.tT_HW_HC_Re.Ai;
	MM2VIS.bHWF_Dem					:=	OUT_HC.tHWF_Dem.Do AND NOT MM2VIS.bMsg2750;
	MM2VIS.bChC_Heating_Dem 		:=  OUT_HC.tChC_Heating.Do;
	MM2VIS.bECW_ShutOffVal_Dem		:=	OUT_HC.tECW_ShutOffVal_Dem.Do;
	MM2VIS.bECW_ShutOffVal_Dem_Exist:=	bECW_ShutOffVal_Dem_Exist;
	MM2VIS.bValHeater_Dem			:=	OUT_HC.tValHeater_Dem.Do;
	MM2VIS.bValHeater_Dem_Exist		:=	bValHeater_Dem_Exist;
	MM2VIS.bFanRingHeater_Dem		:=	OUT_HC.tFanRingHeater_Dem.Do;
	MM2VIS.bFanRingHeater_Dem_Exist	:=	bFanRingHeater_Dem_Exist;

	MM2VIS.bChC2_DemPump		:=	OUT_HC.tChC2_DemPump.Do;
	MM2VIS.iSumChC2_Stages		:=	iSumChC2_Stages;
	MM2VIS.bChC2_On    			:= (MM2VIS.iSumChC2_Stages = 1 AND NOT MM2VIS.bMsg9228) OR (MM2VIS.iSumChC2_Stages > 1 AND MM2VIS.bMsg9228);
	MM2VIS.bChC2_Heating_Dem 	:=  OUT_HC.tChC2_Heating.Do;
	MM2VIS.rT_ChC2_Re_LT		:=  IN_HC.tT_ChC2_Re_LT.Ai;
	MM2VIS.rT_ChC2_Su_LT		:=  IN_HC.tT_ChC2_Su_LT.Ai;

	MM2VIS.rT_HW_Su_Unit		:=	IN_HC.tT_HW_Su_Unit.Ai;		(* SAFETY PLC *)
END_PROGRAM
```

### Program Logical/HeatingCooling/ParHC (IEC, version 4.06.0) - + parameter handling

- perm_par.st (not readable text: treated as protected, skipped)

#### perm_par.var
```iecst
VAR
	tParaIntern : ParaHandler_typ; (*Connector type to perm_par*)
	tMM2ParaBase_ReadBack : MM2ParaBase_type; (*INTERNAL! V4.06 new readback structure for information from previous tasks*)
	bWriteDataObj : BOOL; (* TRUE=write data object module *)
	bDataObjLenErr : BOOL; (*Error occured in permem: data module size missmatch*)
	bCreateDataObj : BOOL; (* TRUE=create new data object *)
	bWriteOnce : BOOL; (* write permanent memory once *)
	DatObjCreate_01 : DatObjCreate; (* data object create *)
	DatObjInfoBak_02 : DatObjInfo; (* data object info *)
	DatObjDelete_01 : DatObjDelete; (* data object delete *)
	DatObjRead_01 : DatObjRead; (* data object read *)
	DatObjRead_02 : DatObjRead; (* manual initiated data object read *)
	DatObjWrite_01 : DatObjWrite; (* data object write *)
	DatObjDelete_02 : DatObjDelete; (* data object delete *)
	DatObjDelete_11 : DatObjDelete; (*Delete Backup File*)
	DatObjInfo_01 : DatObjInfo; (* data object info *)
	DatObjInfo_02 : DatObjInfo; (* data object info *)
	szModuleName : STRING[35]; (* module name of object *)
	szModuleNameBackup : STRING[35]; (* module name of posiibly created backup object *)
	DatObjCopy_01 : DatObjCopy;
	bCopyDataObj : BOOL;
	TON_WarnDelay : TON;
	TON_WritePMEM : TON; (* delay write permanent memory *)
	ulPMPointer : UDINT; (* adress of actual checksum value *)
	ulChecksum : UDINT; (* parameter checksum value *)
	pm_len : UDINT; (* permanent value lenght *)
	ulChecksumOld : UDINT; (* last vlaue of parameter checksum *)
	ulChkValue : UDINT; (* actual value of parameter pointer *)
	pm_id : UDINT; (* permanent value identifier *)
	pm_p : UDINT; (* permanent value pointer *)
	DatObjInfo_META : DatObjInfo;
	DatObjRead_META : DatObjRead;
	szMetaDataRaw : STRING[2000];
	szMetaData : ARRAY[0..4] OF STRING[35];
	szMetaDataVis : ARRAY[0..3] OF STRING[35];
	ssIndex : INT;
	ssCount : INT;
	ucMetaDataRaw : ARRAY[0..2000] OF USINT;
	ssCount2 : INT;
	szMetaDataFile : STRING[10];
	szText1 : STRING[20];
	pv_adr_IN_XX_tPB2MM : UDINT;
	pv_lng : UDINT;
	pv_lng_IN_XX_tPB2MM : UDINT;
	pv_lng_OUT_XX_tPB2MM : UDINT;
	szText2 : STRING[20];
	pv_adr_OUT_XX_tXX2PB : UDINT;
END_VAR
VAR CONSTANT
	ERR_NOERROR : UINT := 0;
END_VAR
VAR
	usPMWriteCnt : UINT;
	pm_Error : UDINT; (* permanent value error *) (* Deleted: pm : ParaMem_typ; permanent memory tags mathias, 22.8.11*)
	fun_Error : UDINT := 0; (*state > 0 = function error*)
	xLocalParaCheck : ParaCheckFUB; (*local function instance to check parameter values*)
	TON_ParaSetupOk : TON;
	bParaCheckSystemOk : BOOL;
	iDebug_ParaOkChecked : UDINT;
	bRestoreBackupDataObj : BOOL := FALSE;
	bRestoreDataObjContent : BOOL := FALSE;
	pm_id_backup : UDINT;
	pm_p_Backup : UDINT;
	DatObjCopy_02 : DatObjCopy;
	bDeleteBackupDataObj : BOOL := FALSE; (*Command to delete backup data module file on purpose*)
	bDebugPara : ARRAY[0..5] OF BOOL;
	ssIndex2 : INT;
	ssIndex3 : INT;
	ssIndex4 : INT;
	ssIndexVis : INT;
	szText : STRING[40];
	pv_adr_Para : UDINT;
	szParaSnippet : ARRAY[0..5] OF STRING[150];
	szParaIndex : STRING[10];
	slValue : DINT;
	iModuleDLD_ResetCount : INT;
	bDownloadDetected : BOOL;
	bFlagParaStructCopyWorking : BOOL; (*true, if cyclic para copying is active, 1 false cycle at every copy *)
	bStoreInitParaInDataObj : BOOL := FALSE;
	bTestflag : BOOL;
	bReadOutMETA_Once : BOOL;
	tParaCheck_iPvAdress : ARRAY[0..5] OF UDINT;
	tParaCheck_iPvLengt : ARRAY[0..5] OF UDINT;
	tParaCheck_rPvValue : ARRAY[0..5] OF REAL;
	tParaCheck_rRangeMIN : ARRAY[0..5] OF REAL;
	tParaCheck_rRangeMAX : ARRAY[0..5] OF REAL;
	tParaCheck_szPvName : ARRAY[0..5] OF STRING[35];
	ssFormatDetected : INT;
	szMetaDataPart : STRING[150];
	szFullTaskName : STRING[35];
	szFullMetaModuleName : STRING[35];
	debugLen : INT;
	debugSize : INT := 0;
	strcat_adr1 : UDINT;
	strcat_adr2 : UDINT;
	ssIndexTN : INT;
	bAlternate : BOOL;
	n : INT;
	iAlternateChecksum : DINT;
	iAlternateChecksumOld : DINT;
	ulDebugChkValue : ARRAY[0..999] OF UDINT;
	Adr1 : UDINT;
	Adr2 : UDINT;
	usPMWriteCntStepsize : UINT := 1; (*different step sizes to help debug*)
	usPMWriteCntXOR : UINT;
	usPMWriteCntAltSum : UINT;
	ulAdrPM : UDINT;
	usChkValuePM : USINT;
	ulAdrPara : UDINT;
	ulPara_len : UDINT;
	usChkValuePara : USINT;
	iDebugCountPMDifferences : DINT := 0;
	bEngineRunDetected : BOOL; (*detection status bit autocommand 100 /101  for engine run state*)
	ucMetaDataDebugInfoLine : ARRAY[0..24] OF STRING[80];
	ssIndexMand : INT := 0;
	szMetaDataMand : STRING[35];
	iMyErrorInfo_Autoreset : DINT; (*internal autoreset counter*)
	ssIndex_Version : INT; (*internal*)
	ssIndex_BU : INT; (*internal*)
	ssIndex_BU2 : INT; (*internal*)
END_VAR
```

### Program Logical/HeatingCooling/PermHC (IEC, version 4.04.0) - + PermanentMemory

- PermHCCyclic.st (not readable text: treated as protected, skipped)

- PermHCInit.st (not readable text: treated as protected, skipped)

#### PermHC.var - Local variables
```iecst
VAR
	pm_Error : UINT;
	write_once : BOOL;
	pm_len : UDINT;
	ModulName : STRING[35];
	DatObjInfo_01 : DatObjInfo;
	pm_id : UDINT;
	pm_p : UDINT;
	bCreateDataObj : BOOL;
	perm_par_vers : UINT;
	DatObjRead_01 : DatObjRead;
	DatObjDelete_PermMem : DatObjDelete;
	DatObjCreate_01 : DatObjCreate;
	DatObjWrite_01 : DatObjWrite;
	ulChecksumOld : UDINT;
	ulPMPointer : UDINT;
	ulChkValue : UDINT;
	TON_WritePMEM : TON;
	ulChecksum : UDINT;
	bWriteDataObj : BOOL;
	TON_WarnDelay : TON;
	TON_BlockMinFileAge : TON; (*waiting time without file write after successful performed write*)
	bBlock_MinFileAge : BOOL := FALSE; (*pause the perm file write after each sucessful write*)
	iPM_WriteCnt : UDINT; (* *) (*old VarName: usPMWriteCnt*)
END_VAR
VAR CONSTANT
	ERR_NOERROR : UINT := 0;
END_VAR
VAR
	pmm : Perm_HC_Struct;
END_VAR
```

### Package Logical/ICxx - IC: Ignition Controller

### Data object Logical/ICxx/META_IC (Simple) - MODUL META data file

#### META_IC.dat
```
; *******************************************************************************
; AGGR: Module Meta Data (data module)
;
; This code is confidential and proprietary to the INNIO Company.
; It may not be used in any form, or reproduced in any manner, without the express
; written permission of the INNIO Company.
; Copyright, INNIO Company, 2024
;
; Customized modifications: -
; ------------------------
;
; History:
; -------
; V03.99.00.00	06.03.2013	Weitzer		generated for modular software
; V03.99.02.00	29.05.2013	Zengerer	initial dependencies prepared
; V04.00.00.00	30.01.2014	Denk		new version
; V04.00.01.00	21.04.2014	Denk		new version
; V04.00.02.00	20.06.2014	Denk		new version
; V04.00.03.00	10.07.2014	Denk		caniniIc: ic900_vis added
; V04.00.04.00	11.12.2014	Denk		Bugfix, missing messages 3052,3209. RiskClass for all alarms checked and corrected.
; V04.00.05.00	15.07.2015	Weitzer		optimizing of speed measurement and MissFire command
; V04.03.00.00	02.11.2015	Zengerer 	MANDATORYMODULE statement
; V04.04.00.00	15.05.2017	Gwiggner 	KLS98 validation - bugfix ignition timing point
; V04.05.00.00	27.07.2017	Messner		CAN Diagnosis Picture added
; V04.07.00.00	23.01.2019	Zengerer	Distribute Para task with perm messaage handling capability to all modules, no functional change to V4.06
; V04.10.00.00	09.03.2021	Andre		Skip fire bug fix
; V04.12.00.00	08.09.2022	Andre		Added changes for SEMIC including new SEMIC task
; V04.13.00.00	17.10.2022	Andre		Added FW 201.22. Fixed issues 1193, 1229, 1248, 1261.
; 				08.03.2024	Andre		Added FW 201.25. Set the output failure rate to 0 during the ignition self-test.
; V04.14.00.00	22.10.2024	Andre		Added 10s timer to generate OUT_IC.bIC_IgnEngergy_Hi
; 				27.11.2024	Andre		Extended maximum time for skip fire during purge starts with skip fire.
; 				18.12.2024	Andre		Send global and individual ITP during full SEMIC configuration.
; 										Avoid rounding issues of the cylinder-specific ITP offset calculation.
; 										Do not set B9049 if A3024 is set. Reset B9049 only when warning missing trigger 1 and 2 are not active.
;				28.01.2025	Andre		Fix potential A2363 after trip prio 1 or 2.
;				07.03.2025	Andre		Avoid W9339 in WinMOD simulation.
;
; Instructions for use:
; --------------------
; make only changes at the version numbers
;
; Outstandings:
; ------------
;
; *******************************************************************************
;
"<META>"
;
; Module ID
"<MODUL>IC</MODUL>"
;
; Module Version (xx.yy.zz.cc)
"<VERSION>04.14.00.00</VERSION>"
;
; Module Basisupdate Version BU (00-99)
"<BASISUPDATE_VERSION>00</BASISUPDATE_VERSION>"
;
; Optional: specify order number for limitated module usage
"<ORDER></ORDER>" ;<!--(optional for restricted customizations; missing statement makes module valid for all orders)-->
;
; Parameter Check <PARAn Name='aAbcdef' MIN='xxx' MAX='yyy' />  (watch for correct spacings and apostrophs!)
"<PARAMETER_CHK>"
"	<PARA1 Name='iEng_Motortype' MIN='208' MAX='920' />"
"	<PARA2 />"
"	<PARA3 />"
"	<PARA4 />"
"	<PARA5 />"
"</PARAMETER_CHK>"
;
; Statement, if engine operation is also allowed without this module (FALSE) or if this module´s parameter check passing is mandatory (TRUE)
"<MANDATORYMODULE>TRUE</MANDATORYMODULE>"
;
; Permanent Datamodule Filenames<!-- enter filenames for counter and INTERNAL parameter only; filename without extention-->
"<DATAMODULES>" ;<!-- optional; mehrere DATAMODULES erlaubt-->
"	<DATAMODULE>par_IC</DATAMODULE>"
"</DATAMODULES>"
;
; Dependencies Modules (MMxx.yy.zz.cc)
"<DEPENDENCIES>"
"	<DEPENDENCY MODULE='AB' VERSION='04.00.00.00' />"
"	<DEPENDENCY MODULE='PB' VERSION='04.00.00.00' />"
"	<DEPENDENCY MODULE='HA' VERSION='04.00.00.00' />"
"	<DEPENDENCY MODULE='IG' VERSION='04.00.00.00' />"
"	<DEPENDENCY MODULE='OP' VERSION='04.00.00.00' />"
"	<DEPENDENCY MODULE='EC' VERSION='04.04.00.00' />"
"   <DEPENDENCY VISVERSION='02.13.00.00' />"			; Dependencies Visualization
"</DEPENDENCIES>"
;
; Module function description
"<MODULEFUNCTION>" ;<!-- short overview documentation of module function; add reference to detailed information, if available-->
"	<General>	"
"	CAN communication to Monic device "
"	</General>	"
""
"	<F1 Name='CAN Communication' LastModified='04.00.00.00'>"
"	Manage and monitor CAN communication to igniton device (IC or MIC or SEMIC).	"
"	</F1>"
"	<F2 Name='Parameter sending' LastModified='04.00.00.00'>"
"	 Send parameters and operation values to the device.	"
"	</F2>"
"	<F3 Name='Error handling' LastModified='04.00.00.00'>"
"	 Forward errors from ignition device to control system. 	"
"	</F3>"
"	<F4 Name='Ignition status' LastModified='04.00.00.00'>"
"	 Read actual ignition status. "
"	</F4>"
"	<F5 Name='System version' LastModified='04.00.00.00'>"
"	 Check hard and software version of ignition system. "
"	</F5>"
"	<F6 Name='Ignition selftest' LastModified='04.00.00.00'>"
"	 Handle ignition system selftest mode. "
"	</F6>"
"	<F7 Name='Ignition Controller firmware updater' LastModified='04.00.00.00'>"
"	 Handle the firmware update of SEMIC via CAN bus. "
"	</F7>"
""
"	<Info>"
"	 V4.0.3.0 task caniniIc, ic900_vis added	"
"    V4.04.00.00 KLS98 validation - bugfix ignition timing point"
"	</Info>"
""
"	<Customized LastModified='4.0.0.0'>	"
"	- Nothing "
"	</Customized>	"
""
"</MODULEFUNCTION>"
;
"</META>"
```

### Module_IC.typ - Module global data types
```iecst
TYPE
	IN_IC_Struct : 	STRUCT
		tAB2IC : AmmBase2MM; (*AMM base to ICxx data transfer*) (*OldName:new PV; Cycle:2;*)
		tAB2IC_TC2 : AmmBase2MM; (*AMM base to ICxx data transfer*) (*OldName:new PV; Cycle:2;*)
		tPB2MM : ParaBase2MM_type; (*Data exchange structure to ParaBase*) (*OldName:new PV; Cycle:5;*)
		bIgn_SelfTest : BOOL; (*switch ignition system to selftest *) (*OldName:GoSelftest; Cycle:5;*)
		bEng_Dem : BOOL; (*module demanded*) (*OldName:M_AGFD; Cycle:5;*)
		iCANIdent : UDINT; (*ID number to check if CAN comm. start up was succesful*) (*OldName:ulCANIdent; Cycle:2;*)
		iCANIdent_TC8 : UDINT; (*ID number to check if CAN comm. start up was succesful*) (*OldName:ulCANIdent; Cycle:2;*)
		iSt_OpMode : UDINT; (*engine operation mode*) (*OldName:StartM,StopM; Cycle:5;*)
		iIdx_OMSS : INT; (*Index of operation mode selector switch 0  OFF, 1  MANUAL, 2  AUTOMATIC, 3 Test (Optional)*) (*OldName:BWS_HA,PROBE; Cycle:5;*)
		rCA_IgnP_Set_TC2 : REAL; (* actual ignition timing setpoint *) (*OldName:W_ZZP ; Cycle:5;*)
		rCA_IgnP_Set : REAL; (* actual ignition timing setpoint *) (*OldName:W_ZZP ; Cycle:5;*)
		rCA_Ign_Act_TC2 : ARRAY[0..24]OF REAL; (* actual cylinder igniton point *) (*OldName:ZZPCyl ; Cycle:5;*)
		rCA_Ign_Act : ARRAY[0..24]OF REAL; (* actual cylinder igniton point *) (*OldName:ZZPCyl ; Cycle:5;*)
		bIgn_Dem : BOOL; (*demand ignition*) (*OldName:ZUEND; Cycle:2;*)
		iMisfCyl : UDINT; (*cylinder misfire parameter *) (*OldName:MissfCyl; Cycle:2 *)
		bSimWinMOD_Active : BOOL; (* WinMode simulation active *) (* OldName:new PV; Cycle:5*)
		rP_Act_Norm_Filt : REAL; (*Actual power related to rP_Nom filtered T=1s*) (*OldName:W_ZZP ; Cycle:5;*)
	END_STRUCT;
	OUT_IC_Struct : 	STRUCT
		tIC2PB : MM2ParaBase_type; (*Data exchange structure to ParaBase*) (*OldName:new PV; Cycle:5;*)
		tIC2AB : MM2AmmBase; (*ICxx module to AMM base data transfer*) (*OldName:new PV; Cycle:5;*)
		tICxx_CanGo : CanDeviceGo; (*Start / Stop CAN communication*) (*OldName:CANDevGo; Cycle:5;*)
		rN_IgnIC_Act : REAL; (*Engine speed measured by ignition IC*) (*OldName:ZDGSpeed; Cycle:1;*)
		b_IgnIC_SelfTestBack : BOOL; (*Feedback: Ignition system is in selftest mode*) (*OldName:GoSelftest; Cycle:5;*)
		iIC900CommErrCount : USINT; (* comm. error counter *)
		iE_IgnStat : USINT; (* events igniton system status *)
		bIC_OperationState : BOOL; (*IC operation state*)
		bIC_IgnEngergy_Hi : BOOL; (*IC Warning Maximum Energy Exceeded*)
		bIC_Ign_Run_CAN : BOOL; (*IC Output ignition active from CAN*)
	END_STRUCT;
	CanDeviceGo : 	STRUCT
		CANDevGo : ARRAY[0..1]OF USINT;
		ECANDevGo : USINT;
	END_STRUCT;
	MM2VIS_Struct : 	STRUCT
		bMsg3310 : BOOL; (*3310 Ignition output spare cylinder xx*) (*OldName:ZDGAUS_A; Cycle:;*)
		bMsg3240 : BOOL; (*3240 Ignition output monitoring cylinder xx *) (*OldName:ZDGAUS_B; Cycle:;*)
		bMsg3410 : BOOL; (*3410 Ignition output spare cylinder xx *) (*OldName:ZDGAUS_W; Cycle:;*)
		iMsg3240 : INT; (*3240 Ignition output spare cylinder xx, cylinder info number*) (*OldName:ucZylZAus; Cycle:;*)
		bMsg3027 : BOOL; (* 3027 Ignition CAM pickup missing *) (*OldName:ZDGCAM; Cycle:;*)
		bMsg3031 : BOOL; (* 3031 Ignition CAN communication failure *) (*OldName:ZDGCAN; Cycle:;*)
		bMsg3029 : BOOL; (* 3029 Ignition CPU failure *) (*OldName:ZDGCPU; Cycle:;*)
		bMsg3052 : BOOL; (* 3052 Wrong type of ignition system *) (*OldName:ZDGFALSCH; Cycle:;*)
		bMsg3209 : BOOL; (* 3209 Ignition setting is forbidden during the engine is running *) (*OldName:ZDGPAR; Cycle:;*)
		bMsg3030 : BOOL; (* 3030 Ignition parameter failure *) (*OldName:ZDGPARAM; Cycle:;*)
		bMsg3026 : BOOL; (* 3026 Ignition reset pickup missing *) (*OldName:ZDGRST; Cycle:;*)
		bMsg3025 : BOOL; (* 3025 Ignition trigger pickup missing *) (*OldName:ZDGTRI; Cycle:;*)
		bMsg3028 : BOOL; (* 3028 Ignition shutoff overspeed *) (*OldName:ZDGUEDZ; Cycle:;*)
		bIgnIC_CylOutFail : ARRAY[0..24]OF BOOL; (* Ignition system cylinder output failure *) (*OldName:IgnOFail; Cycle:;*)
		iIgnIC_VersionSW : INT; (* Ignition system software version *) (*OldName:IgnVers; Cycle:;*)
		iIgnIC_SysTypeHW : INT; (* Hardware type of ignition system  *) (*OldName:usIgnSystem; Cycle:;*)
		rEnergLev : REAL; (*Ignition system energy level % *)
		iCMSinit_IC900_status : INT; (* Ignition Module CMS Init Status *)
		iCMSmain_IC900_status : INT; (* Ignition Module Main CMS Status *)
		iNum_OutFailRate : USINT; (*Ignition controller output failure rate*)
		iTi_IgnOph : UINT; (*Ignition controller operating hours [h]*)
		iNum_SNYear : USINT; (*Serial number: year*)
		iNum_SNWeek : USINT; (*Serial number: week*)
		iNum_SNCnt : USINT; (*Serial number: counter*)
		rU_IC_Trig1 : REAL; (*Trigger 1 pickup peak voltage [V]*)
		rU_IC_Trig2 : REAL; (*Trigger 2 pickup peak voltage [V]*)
		rU_IC_Reset : REAL; (*Reset pickup peak voltage [V]*)
		bMsg9339 : BOOL; (*9339 Wrong ignition controller firmware*)
		bMsg9340 : BOOL; (*9340 Ignition failure trigger pickup*)
		bMsg9341 : BOOL; (*9341 Ignition failure reset pickup*)
		bMsg9342 : BOOL; (*9342 Ignition failure cam pickup*)
		bMsg9343 : BOOL; (*9343 Pickup degradation*)
		bMsg9049 : BOOL; (*9049 Ignition failure trigger pickup*)
		iMsg9049 : INT; (*9049 Ignition failure trigger pickup - info*)
		bMsg9315 : BOOL; (*9315 Ignition controller input voltage too low*)
		bMsg2363 : BOOL; (*2363 Ignition controller hardware failure*)
		bMsg2764 : BOOL; (*2764 Ignition controller temperature too high*)
		bMsg2767 : BOOL; (*2767 Wrong pickup polarity*)
		bIC_UnkEngAppCode : BOOL; (*Unknown engine application code*)
		bIC_CfgOoRange : BOOL; (*Configuration out of range*)
		bIC_UnkITP_ELvl : BOOL; (*Unknown global timing or energy level*)
		bIC_ITP_ELvlOoRange : BOOL; (*Global, individual timing or energy level out of range*)
		bIC_E2PROMErr : BOOL; (*E2PROM checksum error*)
		bIC_HwErr : BOOL; (*Hardware error*)
		bIC_OutHarnessErr : BOOL; (*Output harness error*)
		bIC_Overtemp : BOOL; (*Overtemperature*)
		bIC_DOFail : BOOL; (*Digital output failure*)
		rT_IC : REAL; (*Ignition controller temperature [degC]*)
		iE_PrimEnergy : ARRAY[0..24]OF UINT; (*Primary energy demand [mJ]*)
		iE_PrimEnergy_Min : UINT; (*Minimum primary energy demand [mJ]*)
		iE_PrimEnergy_Max : UINT; (*Maximum primary energy demand [mJ]*)
		iE_PrimEnergy_Avg : UINT; (*Average primary energy demand [mJ]*)
		iNum_PUMode : USINT; (*Pickup mode detected by SEMIC*)
		iNum_IC_NrTeethErr : UINT; (*Number of teeth at pickup error*)
		rNum_IcUpdProgress : REAL; (*IC updater progress bar*)
		rNum_SemicFw : REAL; (*SEMIC firmware available for download*)
		bIC_U_PuRes_Lo : BOOL; (*Reset pickup signal too low*)
		bIC_U_PuTrg1_Lo : BOOL; (*Trigger 1 pickup signal too low*)
		bIC_IgnEnaFail : BOOL; (*Ignition enable failure*)
		bIC_U_PuTrg2_Lo : BOOL; (*Trigger 2 pickup signal too low*)
		bIC_PolTrg1 : BOOL; (*Wrong polarity trigger 1 pickup signal*)
		bIC_PolTrg2 : BOOL; (*Wrong polarity trigger 2 pickup signal*)
		bIC_PolRes : BOOL; (*Wrong polarity reset pickup signal*)
		bMsg2367 : BOOL; (*2367 - Wrong or missing ignition coil*)
		bMsg9073 : BOOL; (*9073 - Wrong or missing ignition coil*)
		iMsg9073 : INT; (*9073 - Wrong or missing ignition coil - Cylinder info number*)
		bMsg2375 : BOOL; (*2375 - Ignition coil or wiring failure*)
	END_STRUCT;
	VIS2MM_Struct : 	STRUCT
		bIC_UpdStart : BOOL; (*IC updater start/stop button*)
	END_STRUCT;
	tZDGSpeed : 	STRUCT
		ICSpdAvg : UINT; (*Average engine speed from ignition controller [rpm]*)
		ICSpd16Teeth : UINT; (*16-teeth engine speed from ignition controller [rpm]*)
		ICSpdSPAx : UINT; (*SPAx engine speed from ignition controller [rpm * 10]*)
		ICSpd4Teeth : UINT; (*4-teeth engine speed from ignition controller [rpm]*)
	END_STRUCT;
	IC_FiringDist : 	STRUCT
		DistOddToEven : UINT; (*Firing distance odd to even output [degCA*10]*)
		DistEvenToOdd : UINT; (*Firing distance even to odd output [degCA*10]*)
	END_STRUCT;
	IC_Curr : 	STRUCT
		Current : UINT; (*Ignition pulse step current [%]*)
		Duration : UINT; (*Ignition pulse step duration*)
	END_STRUCT;
	IC_CoilPara : 	STRUCT
		TimeToPeak : UINT; (*Time to peak voltage [us]*)
		CoilCurrMax : USINT; (*Maximum primary coil current [A]*)
		IgnEnergyMax : UINT; (*Maximum energy for firing event [mJ]*)
	END_STRUCT;
	IC_SpDur : 	STRUCT
		SpDur : UINT; (*Spark duration [us]*)
		SpDurMin : USINT; (*Minimum spark duration [%]*)
	END_STRUCT;
	IC_SpdST : 	STRUCT
		Spd_SelfTest : UINT; (*Speed for self-test [rpm]*)
		TiSTSpdRamp : UINT; (*Selft-test speed ramp-up / down time [s*10]*)
	END_STRUCT;
	IC_U_Pickups : 	STRUCT
		U_Trigger1 : UINT; (*Trigger 1 pickup peak voltage [V*10]*)
		U_Trigger2 : UINT; (*Trigger 2 pickup peak voltage [V*10]*)
		U_Reset : UINT; (*Reset pickup peak voltage [V*10]*)
	END_STRUCT;
	IC_SpInfo : 	STRUCT
		Voltage : UINT; (*Spark voltage [kV*10]*)
		PrimEnergy : UINT; (*Primary energy demand [mJ]*)
	END_STRUCT;
	IC_PUNoiseRate : 	STRUCT
		Trigger1 : USINT; (*Trigger 1 pickup noise rate [1/s]*)
		Trigger2 : USINT; (*Trigger 2 pickup noise rate [1/s]*)
		Reset : USINT; (*Reset pickup noise rate [1/s]*)
		Cam : USINT; (*CAM pickup noise rate [1/s]*)
		TRIGGER : USINT; (*TRG pickup noise rate [1/s]*)
		CAMRESET : USINT; (*C/R pickup noise rate [1/s]*)
	END_STRUCT;
	IC_PrimEnergyStat : 	STRUCT
		PrimEnergyMin : UINT; (*Minimum primary energy demand [mJ]*)
		PrimEnergyAvg : UINT; (*Avergae primary energy demand [mJ]*)
		PrimEnergyMax : UINT; (*Maximum primary energy demand [mJ]*)
	END_STRUCT;
	CoilParam : 	STRUCT
		data1 : USINT;
		data2 : USINT;
		data3 : USINT;
		data4 : USINT;
		data5 : USINT;
		data6 : USINT;
	END_STRUCT;
	CoilParam5 : 	STRUCT
		data1 : USINT;
		data2 : USINT;
		data3 : USINT;
		data4 : USINT;
		data5 : USINT;
	END_STRUCT;
	CoilParam6 : 	STRUCT
		data1 : USINT;
		data2 : USINT;
	END_STRUCT;
	IC_CurrPmmReal : 	STRUCT
		Current : REAL;
		Time : REAL;
	END_STRUCT;
END_TYPE
```
